LIN {X 0.236,Y -556.515,Z 1541.490,A 0.000,B 0.000,C 90.000,E1 124.199} C_DIS
LIN {X 0.231,Y -556.880,Z 1541.484,A 0.000,B 0.000,C 90.000,E1 123.086} C_DIS
LIN {X -0.003,Y -557.168,Z 1541.476,A 0.000,B 0.000,C 90.000,E1 121.720} C_DIS
LIN {X 0.132,Y -557.913,Z 1541.462,A 0.000,B 0.000,C 90.000,E1 119.205} C_DIS
LIN {X 0.047,Y -558.358,Z 1541.456,A 0.000,B 0.000,C 90.000,E1 118.103} C_DIS
LIN {X 0.056,Y -558.863,Z 1541.447,A 0.000,B 0.000,C 90.000,E1 116.437} C_DIS
LIN {X -0.021,Y -559.208,Z 1541.441,A 0.000,B 0.000,C 90.000,E1 115.335} C_DIS
LIN {X -0.037,Y -559.617,Z 1541.433,A 0.000,B 0.000,C 90.000,E1 113.951} C_DIS
LIN {X -0.269,Y -559.870,Z 1541.425,A 0.000,B 0.000,C 90.000,E1 112.589} C_DIS
LIN {X 0.126,Y -560.109,Z 1541.415,A 0.000,B 0.000,C 90.000,E1 110.610} C_DIS
LIN {X 0.134,Y -560.466,Z 1541.404,A 0.000,B 0.000,C 90.000,E1 108.671} C_DIS
LIN {X 0.145,Y -560.782,Z 1541.393,A 0.000,B 0.000,C 90.000,E1 106.732} C_DIS
LIN {X -0.026,Y -561.131,Z 1541.381,A 0.000,B 0.000,C 90.000,E1 104.537} C_DIS
LIN {X -0.171,Y -561.673,Z 1541.367,A 0.000,B 0.000,C 90.000,E1 102.063} C_DIS
LIN {X 0.022,Y -562.418,Z 1541.353,A 0.000,B 0.000,C 90.000,E1 99.557} C_DIS
LIN {X 0.312,Y -562.996,Z 1541.344,A 0.000,B 0.000,C 90.000,E1 97.871} C_DIS
LIN {X -0.187,Y -563.479,Z 1541.336,A 0.000,B 0.000,C 90.000,E1 96.543} C_DIS
LIN {X -0.081,Y -564.062,Z 1541.327,A 0.000,B 0.000,C 90.000,E1 94.878} C_DIS
LIN {X -0.053,Y -564.429,Z 1541.319,A 0.000,B 0.000,C 90.000,E1 93.498} C_DIS
LIN {X 0.057,Y -564.999,Z 1541.310,A 0.000,B 0.000,C 90.000,E1 91.835} C_DIS
LIN {X -0.161,Y -565.788,Z 1541.298,A 0.000,B 0.000,C 90.000,E1 89.656} C_DIS
LIN {X -0.247,Y -566.843,Z 1541.284,A 0.000,B 0.000,C 90.000,E1 87.192} C_DIS
LIN {X 0.050,Y -567.682,Z 1541.274,A 0.000,B 0.000,C 90.000,E1 85.241} C_DIS
LIN {X -0.107,Y -569.181,Z 1541.257,A 0.000,B 0.000,C 90.000,E1 82.243} C_DIS
LIN {X 0.052,Y -570.789,Z 1541.245,A 0.000,B 0.000,C 90.000,E1 80.038} C_DIS
LIN {X -0.035,Y -572.121,Z 1541.236,A 0.000,B 0.000,C 90.000,E1 78.409} C_DIS
LIN {X -0.018,Y -573.750,Z 1541.224,A 0.000,B 0.000,C 90.000,E1 76.228} C_DIS
LIN {X 0.006,Y -574.797,Z 1541.216,A 0.000,B 0.000,C 90.000,E1 74.866} C_DIS
LIN {X 0.042,Y -575.718,Z 1541.208,A 0.000,B 0.000,C 90.000,E1 73.504} C_DIS
LIN {X -0.285,Y -576.881,Z 1541.198,A 0.000,B 0.000,C 90.000,E1 71.638} C_DIS
LIN {X -0.015,Y -578.115,Z 1541.186,A 0.000,B 0.000,C 90.000,E1 69.444} C_DIS
LIN {X 0.256,Y -579.057,Z 1541.177,A 0.000,B 0.000,C 90.000,E1 67.794} C_DIS
LIN {X 0.079,Y -580.085,Z 1541.166,A 0.000,B 0.000,C 90.000,E1 65.921} C_DIS
LIN {X 0.030,Y -581.371,Z 1541.154,A 0.000,B 0.000,C 90.000,E1 63.768} C_DIS
LIN {X 0.017,Y -582.452,Z 1541.145,A 0.000,B 0.000,C 90.000,E1 62.153} C_DIS
LIN {X 0.153,Y -583.335,Z 1541.138,A 0.000,B 0.000,C 90.000,E1 60.795} C_DIS
LIN {X 0.080,Y -584.189,Z 1541.130,A 0.000,B 0.000,C 90.000,E1 59.459} C_DIS
LIN {X 0.028,Y -585.143,Z 1541.123,A 0.000,B 0.000,C 90.000,E1 58.122} C_DIS
LIN {X -0.019,Y -586.054,Z 1541.115,A 0.000,B 0.000,C 90.000,E1 56.786} C_DIS
LIN {X -0.084,Y -586.770,Z 1541.110,A 0.000,B 0.000,C 90.000,E1 55.722} C_DIS
LIN {X -0.271,Y -587.524,Z 1541.102,A 0.000,B 0.000,C 90.000,E1 54.402} C_DIS
LIN {X -0.107,Y -588.020,Z 1541.095,A 0.000,B 0.000,C 90.000,E1 53.050} C_DIS
LIN {X -0.203,Y -588.474,Z 1541.086,A 0.000,B 0.000,C 90.000,E1 51.457} C_DIS
LIN {X 0.134,Y -588.756,Z 1541.080,A 0.000,B 0.000,C 90.000,E1 50.356} C_DIS
LIN {X 0.273,Y -588.760,Z 1541.075,A 0.000,B 0.000,C 90.000,E1 49.542} C_DIS
LIN {X 0.215,Y -588.563,Z 1541.073,A 0.000,B 0.000,C 90.000,E1 49.013} C_DIS
LIN {X 0.155,Y -588.189,Z 1541.069,A 0.000,B 0.000,C 90.000,E1 48.485} C_DIS
LIN {X -0.095,Y -587.881,Z 1541.068,A 0.000,B 0.000,C 90.000,E1 48.243} C_DIS
LIN {X -0.160,Y -586.881,Z 1541.065,A 0.000,B 0.000,C 90.000,E1 47.715} C_DIS
LIN {X -0.014,Y -586.191,Z 1541.064,A 0.000,B 0.000,C 90.000,E1 47.433} C_DIS
LIN {X 0.165,Y -585.154,Z 1541.062,A 0.000,B 0.000,C 90.000,E1 47.148} C_DIS
LIN {X 0.054,Y -584.440,Z 1541.061,A 0.000,B 0.000,C 90.000,E1 47.025} C_DIS
LIN {X 0.031,Y -583.064,Z 1541.060,A 0.000,B 0.000,C 90.000,E1 46.863} C_DIS
LIN {X 0.138,Y -582.631,Z 1541.060,A 0.000,B 0.000,C 90.000,E1 46.824} C_DIS
LIN {X -0.118,Y -581.797,Z 1541.060,A 0.000,B 0.000,C 90.000,E1 46.824} C_DIS
LIN {X -0.127,Y -422.308,Z 1541.060,A 0.000,B 0.000,C 90.000,E1 46.824} C_DIS
LIN {X 0.122,Y -418.840,Z 1541.050,A 0.000,B 0.000,C 90.000,E1 44.919} C_DIS
LIN {X -0.221,Y -416.461,Z 1541.044,A 0.000,B 0.000,C 90.000,E1 43.947} C_DIS
LIN {X 0.118,Y -407.450,Z 1541.019,A 0.000,B 0.000,C 90.000,E1 39.439} C_DIS
LIN {X 0.243,Y -405.717,Z 1541.013,A 0.000,B 0.000,C 90.000,E1 38.382} C_DIS
LIN {X 0.206,Y -397.431,Z 1540.990,A 0.000,B 0.000,C 90.000,E1 34.199} C_DIS
LIN {X 0.070,Y -393.663,Z 1540.976,A 0.000,B 0.000,C 90.000,E1 31.750} C_DIS
LIN {X -0.160,Y -386.269,Z 1540.953,A 0.000,B 0.000,C 90.000,E1 27.513} C_DIS
LIN {X -0.001,Y -383.047,Z 1540.939,A 0.000,B 0.000,C 90.000,E1 24.975} C_DIS
LIN {X -0.032,Y -381.933,Z 1540.935,A 0.000,B 0.000,C 90.000,E1 24.259} C_DIS
LIN {X 0.090,Y -375.539,Z 1540.909,A 0.000,B 0.000,C 90.000,E1 19.523} C_DIS
LIN {X 0.085,Y -373.444,Z 1540.896,A 0.000,B 0.000,C 90.000,E1 17.330} C_DIS
LIN {X 0.018,Y -367.914,Z 1540.868,A 0.000,B 0.000,C 90.000,E1 12.187} C_DIS
LIN {X 0.037,Y -366.509,Z 1540.855,A 0.000,B 0.000,C 90.000,E1 9.962} C_DIS
LIN {X -0.027,Y -361.808,Z 1540.822,A 0.000,B 0.000,C 90.000,E1 4.012} C_DIS
LIN {X -0.142,Y -360.904,Z 1540.802,A 0.000,B 0.000,C 90.000,E1 0.286} C_DIS
LIN {X -0.053,Y -359.426,Z 1540.770,A 0.000,B 0.000,C 90.000,E1 354.546} C_DIS
LIN {X 0.070,Y -358.890,Z 1540.759,A 0.000,B 0.000,C 90.000,E1 352.648} C_DIS
LIN {X -0.020,Y -359.563,Z 1540.726,A 0.000,B 0.000,C 90.000,E1 346.645} C_DIS
LIN {X 0.001,Y -361.801,Z 1540.684,A 0.000,B 0.000,C 90.000,E1 339.135} C_DIS
LIN {X -0.154,Y -362.053,Z 1540.680,A 0.000,B 0.000,C 90.000,E1 338.411} C_DIS
LIN {X 0.189,Y -365.980,Z 1540.643,A 0.000,B 0.000,C 90.000,E1 331.641} C_DIS
LIN {X 0.029,Y -366.387,Z 1540.639,A 0.000,B 0.000,C 90.000,E1 330.923} C_DIS
LIN {X -0.031,Y -371.355,Z 1540.604,A 0.000,B 0.000,C 90.000,E1 324.642} C_DIS
LIN {X -0.043,Y -371.766,Z 1540.602,A 0.000,B 0.000,C 90.000,E1 324.276} C_DIS
LIN {X 0.013,Y -377.358,Z 1540.567,A 0.000,B 0.000,C 90.000,E1 318.038} C_DIS
LIN {X 0.012,Y -378.235,Z 1540.563,A 0.000,B 0.000,C 90.000,E1 317.310} C_DIS
LIN {X 0.002,Y -383.940,Z 1540.531,A 0.000,B 0.000,C 90.000,E1 311.515} C_DIS
LIN {X 0.088,Y -384.893,Z 1540.527,A 0.000,B 0.000,C 90.000,E1 310.782} C_DIS
LIN {X 0.262,Y -390.610,Z 1540.495,A 0.000,B 0.000,C 90.000,E1 305.025} C_DIS
LIN {X 0.106,Y -391.104,Z 1540.493,A 0.000,B 0.000,C 90.000,E1 304.692} C_DIS
LIN {X 0.022,Y -391.648,Z 1540.489,A 0.000,B 0.000,C 90.000,E1 303.992} C_DIS
LIN {X -0.080,Y -396.825,Z 1540.459,A 0.000,B 0.000,C 90.000,E1 298.693} C_DIS
LIN {X -0.210,Y -397.120,Z 1540.457,A 0.000,B 0.000,C 90.000,E1 298.359} C_DIS
LIN {X -0.055,Y -401.597,Z 1540.426,A 0.000,B 0.000,C 90.000,E1 292.717} C_DIS
LIN {X 0.222,Y -404.659,Z 1540.395,A 0.000,B 0.000,C 90.000,E1 287.094} C_DIS
LIN {X -0.079,Y -404.735,Z 1540.391,A 0.000,B 0.000,C 90.000,E1 286.441} C_DIS
LIN {X 0.214,Y -406.099,Z 1540.364,A 0.000,B 0.000,C 90.000,E1 281.535} C_DIS
LIN {X -0.176,Y -406.094,Z 1540.362,A 0.000,B 0.000,C 90.000,E1 281.243} C_DIS
LIN {X -0.097,Y -405.680,Z 1540.333,A 0.000,B 0.000,C 90.000,E1 276.024} C_DIS
LIN {X -0.165,Y -405.058,Z 1540.328,A 0.000,B 0.000,C 90.000,E1 274.992} C_DIS
LIN {X -0.060,Y -403.497,Z 1540.304,A 0.000,B 0.000,C 90.000,E1 270.802} C_DIS
LIN {X -0.092,Y -403.288,Z 1540.302,A 0.000,B 0.000,C 90.000,E1 270.458} C_DIS
LIN {X 0.091,Y -398.931,Z 1540.271,A 0.000,B 0.000,C 90.000,E1 264.837} C_DIS
LIN {X -0.040,Y -393.108,Z 1540.242,A 0.000,B 0.000,C 90.000,E1 259.567} C_DIS
LIN {X -0.079,Y -392.835,Z 1540.240,A 0.000,B 0.000,C 90.000,E1 259.218} C_DIS
LIN {X 0.034,Y -385.993,Z 1540.212,A 0.000,B 0.000,C 90.000,E1 254.212} C_DIS
LIN {X -0.026,Y -385.267,Z 1540.208,A 0.000,B 0.000,C 90.000,E1 253.504} C_DIS
LIN {X -0.004,Y -384.768,Z 1540.206,A 0.000,B 0.000,C 90.000,E1 253.142} C_DIS
LIN {X 0.221,Y -377.973,Z 1540.182,A 0.000,B 0.000,C 90.000,E1 248.773} C_DIS
LIN {X -0.044,Y -376.233,Z 1540.174,A 0.000,B 0.000,C 90.000,E1 247.358} C_DIS
LIN {X 0.057,Y -374.944,Z 1540.170,A 0.000,B 0.000,C 90.000,E1 246.613} C_DIS
LIN {X -0.208,Y -368.417,Z 1540.148,A 0.000,B 0.000,C 90.000,E1 242.615} C_DIS
LIN {X 0.097,Y -366.047,Z 1540.137,A 0.000,B 0.000,C 90.000,E1 240.717} C_DIS
LIN {X 0.004,Y -359.196,Z 1540.115,A 0.000,B 0.000,C 90.000,E1 236.628} C_DIS
LIN {X 0.021,Y -355.842,Z 1540.100,A 0.000,B 0.000,C 90.000,E1 233.989} C_DIS
LIN {X -0.173,Y -348.793,Z 1540.075,A 0.000,B 0.000,C 90.000,E1 229.461} C_DIS
LIN {X -0.097,Y -346.185,Z 1540.062,A 0.000,B 0.000,C 90.000,E1 227.148} C_DIS
LIN {X -0.088,Y -345.065,Z 1540.058,A 0.000,B 0.000,C 90.000,E1 226.377} C_DIS
LIN {X 0.094,Y -338.586,Z 1540.030,A 0.000,B 0.000,C 90.000,E1 221.310} C_DIS
LIN {X 0.094,Y -336.840,Z 1540.019,A 0.000,B 0.000,C 90.000,E1 219.358} C_DIS
LIN {X 0.014,Y -330.861,Z 1539.988,A 0.000,B 0.000,C 90.000,E1 213.865} C_DIS
LIN {X 0.149,Y -329.296,Z 1539.975,A 0.000,B 0.000,C 90.000,E1 211.465} C_DIS
LIN {X -0.154,Y -324.669,Z 1539.942,A 0.000,B 0.000,C 90.000,E1 205.540} C_DIS
LIN {X 0.174,Y -323.837,Z 1539.928,A 0.000,B 0.000,C 90.000,E1 203.078} C_DIS
LIN {X -0.017,Y -321.124,Z 1539.881,A 0.000,B 0.000,C 90.000,E1 194.662} C_DIS
LIN {X 0.138,Y -320.932,Z 1539.877,A 0.000,B 0.000,C 90.000,E1 193.828} C_DIS
LIN {X -0.076,Y -321.562,Z 1539.832,A 0.000,B 0.000,C 90.000,E1 185.796} C_DIS
LIN {X -0.143,Y -324.415,Z 1539.790,A 0.000,B 0.000,C 90.000,E1 178.165} C_DIS
LIN {X -0.141,Y -325.376,Z 1539.783,A 0.000,B 0.000,C 90.000,E1 176.963} C_DIS
LIN {X -0.100,Y -329.112,Z 1539.750,A 0.000,B 0.000,C 90.000,E1 170.971} C_DIS
LIN {X 0.061,Y -334.260,Z 1539.726,A 0.000,B 0.000,C 90.000,E1 166.589} C_DIS
LIN {X 0.067,Y -335.488,Z 1539.719,A 0.000,B 0.000,C 90.000,E1 165.408} C_DIS
LIN {X 0.143,Y -340.932,Z 1539.695,A 0.000,B 0.000,C 90.000,E1 161.094} C_DIS
LIN {X -0.172,Y -342.138,Z 1539.691,A 0.000,B 0.000,C 90.000,E1 160.369} C_DIS
LIN {X -0.058,Y -347.939,Z 1539.667,A 0.000,B 0.000,C 90.000,E1 156.102} C_DIS
LIN {X -0.081,Y -354.259,Z 1539.648,A 0.000,B 0.000,C 90.000,E1 152.666} C_DIS
LIN {X -0.222,Y -361.406,Z 1539.625,A 0.000,B 0.000,C 90.000,E1 148.535} C_DIS
LIN {X 0.065,Y -368.758,Z 1539.606,A 0.000,B 0.000,C 90.000,E1 145.135} C_DIS
LIN {X 0.065,Y -377.029,Z 1539.584,A 0.000,B 0.000,C 90.000,E1 141.090} C_DIS
LIN {X -0.061,Y -383.435,Z 1539.570,A 0.000,B 0.000,C 90.000,E1 138.566} C_DIS
LIN {X -0.015,Y -385.037,Z 1539.566,A 0.000,B 0.000,C 90.000,E1 137.838} C_DIS
LIN {X -0.004,Y -394.325,Z 1539.544,A 0.000,B 0.000,C 90.000,E1 133.905} C_DIS
LIN {X 0.107,Y -399.276,Z 1539.534,A 0.000,B 0.000,C 90.000,E1 132.123} C_DIS
LIN {X 0.210,Y -400.192,Z 1539.532,A 0.000,B 0.000,C 90.000,E1 131.757} C_DIS
LIN {X 0.078,Y -404.788,Z 1539.521,A 0.000,B 0.000,C 90.000,E1 129.806} C_DIS
LIN {X 0.058,Y -545.511,Z 1539.521,A 0.000,B 0.000,C 90.000,E1 129.806} C_DIS
LIN {X 0.013,Y -547.395,Z 1539.521,A 0.000,B 0.000,C 90.000,E1 129.688} C_DIS
LIN {X 0.033,Y -548.800,Z 1539.519,A 0.000,B 0.000,C 90.000,E1 129.483} C_DIS
LIN {X 0.077,Y -550.101,Z 1539.518,A 0.000,B 0.000,C 90.000,E1 129.197} C_DIS
LIN {X 0.131,Y -551.079,Z 1539.516,A 0.000,B 0.000,C 90.000,E1 128.910} C_DIS
LIN {X -0.186,Y -552.562,Z 1539.513,A 0.000,B 0.000,C 90.000,E1 128.382} C_DIS
LIN {X -0.060,Y -553.654,Z 1539.510,A 0.000,B 0.000,C 90.000,E1 127.810} C_DIS
LIN {X 0.151,Y -554.899,Z 1539.505,A 0.000,B 0.000,C 90.000,E1 126.950} C_DIS
LIN {X -0.074,Y -555.742,Z 1539.501,A 0.000,B 0.000,C 90.000,E1 126.137} C_DIS
LIN {X -0.093,Y -556.443,Z 1539.495,A 0.000,B 0.000,C 90.000,E1 125.025} C_DIS
LIN {X -0.100,Y -556.919,Z 1539.488,A 0.000,B 0.000,C 90.000,E1 123.913} C_DIS
LIN {X -0.177,Y -557.170,Z 1539.484,A 0.000,B 0.000,C 90.000,E1 123.086} C_DIS
LIN {X 0.067,Y -557.444,Z 1539.476,A 0.000,B 0.000,C 90.000,E1 121.671} C_DIS
LIN {X -0.049,Y -558.086,Z 1539.464,A 0.000,B 0.000,C 90.000,E1 119.461} C_DIS
LIN {X -0.344,Y -558.601,Z 1539.456,A 0.000,B 0.000,C 90.000,E1 118.103} C_DIS
LIN {X -0.081,Y -559.095,Z 1539.447,A 0.000,B 0.000,C 90.000,E1 116.411} C_DIS
LIN {X -0.103,Y -559.429,Z 1539.439,A 0.000,B 0.000,C 90.000,E1 115.027} C_DIS
LIN {X 0.094,Y -559.808,Z 1539.433,A 0.000,B 0.000,C 90.000,E1 113.898} C_DIS
LIN {X 0.086,Y -560.052,Z 1539.425,A 0.000,B 0.000,C 90.000,E1 112.514} C_DIS
LIN {X -0.246,Y -560.313,Z 1539.414,A 0.000,B 0.000,C 90.000,E1 110.610} C_DIS
LIN {X 0.170,Y -560.599,Z 1539.405,A 0.000,B 0.000,C 90.000,E1 108.906} C_DIS
LIN {X 0.018,Y -560.882,Z 1539.394,A 0.000,B 0.000,C 90.000,E1 106.985} C_DIS
LIN {X 0.111,Y -561.151,Z 1539.385,A 0.000,B 0.000,C 90.000,E1 105.315} C_DIS
LIN {X -0.235,Y -561.332,Z 1539.379,A 0.000,B 0.000,C 90.000,E1 104.245} C_DIS
LIN {X 0.026,Y -561.875,Z 1539.367,A 0.000,B 0.000,C 90.000,E1 102.007} C_DIS
LIN {X 0.073,Y -562.531,Z 1539.354,A 0.000,B 0.000,C 90.000,E1 99.792} C_DIS
LIN {X -0.185,Y -563.140,Z 1539.345,A 0.000,B 0.000,C 90.000,E1 98.163} C_DIS
LIN {X -0.118,Y -563.647,Z 1539.338,A 0.000,B 0.000,C 90.000,E1 96.777} C_DIS
LIN {X 0.148,Y -564.314,Z 1539.327,A 0.000,B 0.000,C 90.000,E1 94.821} C_DIS
LIN {X 0.182,Y -564.691,Z 1539.319,A 0.000,B 0.000,C 90.000,E1 93.440} C_DIS
LIN {X -0.249,Y -565.309,Z 1539.310,A 0.000,B 0.000,C 90.000,E1 91.833} C_DIS
LIN {X 0.089,Y -566.099,Z 1539.298,A 0.000,B 0.000,C 90.000,E1 89.599} C_DIS
LIN {X -0.102,Y -567.043,Z 1539.286,A 0.000,B 0.000,C 90.000,E1 87.421} C_DIS
LIN {X 0.093,Y -567.784,Z 1539.276,A 0.000,B 0.000,C 90.000,E1 85.755} C_DIS
LIN {X 0.188,Y -568.369,Z 1539.269,A 0.000,B 0.000,C 90.000,E1 84.375} C_DIS
LIN {X -0.212,Y -569.746,Z 1539.255,A 0.000,B 0.000,C 90.000,E1 81.951} C_DIS
LIN {X 0.060,Y -570.688,Z 1539.248,A 0.000,B 0.000,C 90.000,E1 80.557} C_DIS
LIN {X 0.160,Y -571.581,Z 1539.242,A 0.000,B 0.000,C 90.000,E1 79.454} C_DIS
LIN {X -0.107,Y -572.670,Z 1539.234,A 0.000,B 0.000,C 90.000,E1 78.117} C_DIS
LIN {X 0.283,Y -574.137,Z 1539.223,A 0.000,B 0.000,C 90.000,E1 76.172} C_DIS
LIN {X -0.244,Y -575.166,Z 1539.216,A 0.000,B 0.000,C 90.000,E1 74.866} C_DIS
LIN {X -0.201,Y -576.106,Z 1539.208,A 0.000,B 0.000,C 90.000,E1 73.504} C_DIS
LIN {X 0.028,Y -577.285,Z 1539.198,A 0.000,B 0.000,C 90.000,E1 71.583} C_DIS
LIN {X 0.303,Y -578.536,Z 1539.186,A 0.000,B 0.000,C 90.000,E1 69.390} C_DIS
LIN {X -0.107,Y -579.584,Z 1539.175,A 0.000,B 0.000,C 90.000,E1 67.539} C_DIS
LIN {X -0.267,Y -580.591,Z 1539.165,A 0.000,B 0.000,C 90.000,E1 65.665} C_DIS
LIN {X -0.166,Y -581.736,Z 1539.154,A 0.000,B 0.000,C 90.000,E1 63.768} C_DIS
LIN {X 0.213,Y -583.011,Z 1539.144,A 0.000,B 0.000,C 90.000,E1 61.847} C_DIS
LIN {X -0.002,Y -584.073,Z 1539.135,A 0.000,B 0.000,C 90.000,E1 60.255} C_DIS
LIN {X -0.318,Y -585.347,Z 1539.124,A 0.000,B 0.000,C 90.000,E1 58.408} C_DIS
LIN {X -0.046,Y -586.280,Z 1539.117,A 0.000,B 0.000,C 90.000,E1 57.041} C_DIS
LIN {X 0.243,Y -587.178,Z 1539.109,A 0.000,B 0.000,C 90.000,E1 55.674} C_DIS
LIN {X 0.055,Y -587.940,Z 1539.102,A 0.000,B 0.000,C 90.000,E1 54.356} C_DIS
LIN {X -0.251,Y -588.459,Z 1539.095,A 0.000,B 0.000,C 90.000,E1 53.050} C_DIS
LIN {X 0.122,Y -588.912,Z 1539.086,A 0.000,B 0.000,C 90.000,E1 51.412} C_DIS
LIN {X 0.149,Y -589.505,Z 1539.075,A 0.000,B 0.000,C 90.000,E1 49.542} C_DIS
LIN {X -0.153,Y -589.553,Z 1539.071,A 0.000,B 0.000,C 90.000,E1 48.771} C_DIS
LIN {X -0.205,Y -589.384,Z 1539.068,A 0.000,B 0.000,C 90.000,E1 48.243} C_DIS
LIN {X 0.327,Y -588.608,Z 1539.063,A 0.000,B 0.000,C 90.000,E1 47.391} C_DIS
LIN {X -0.165,Y -587.628,Z 1539.061,A 0.000,B 0.000,C 90.000,E1 46.905} C_DIS
LIN {X 0.016,Y -587.021,Z 1539.059,A 0.000,B 0.000,C 90.000,E1 46.620} C_DIS
LIN {X -0.233,Y -586.190,Z 1539.058,A 0.000,B 0.000,C 90.000,E1 46.377} C_DIS
LIN {X 0.344,Y -584.929,Z 1539.056,A 0.000,B 0.000,C 90.000,E1 46.053} C_DIS
LIN {X -0.274,Y -583.866,Z 1539.055,A 0.000,B 0.000,C 90.000,E1 45.972} C_DIS
LIN {X -0.132,Y -582.963,Z 1539.055,A 0.000,B 0.000,C 90.000,E1 45.891} C_DIS
LIN {X -0.362,Y -582.214,Z 1539.055,A 0.000,B 0.000,C 90.000,E1 45.891} C_DIS
LIN {X 0.017,Y -420.475,Z 1539.055,A 0.000,B 0.000,C 90.000,E1 45.850} C_DIS
LIN {X 0.032,Y -418.598,Z 1539.049,A 0.000,B 0.000,C 90.000,E1 44.798} C_DIS
LIN {X -0.163,Y -409.032,Z 1539.024,A 0.000,B 0.000,C 90.000,E1 40.378} C_DIS
LIN {X 0.020,Y -406.094,Z 1539.015,A 0.000,B 0.000,C 90.000,E1 38.624} C_DIS
LIN {X -0.124,Y -403.870,Z 1539.009,A 0.000,B 0.000,C 90.000,E1 37.604} C_DIS
LIN {X -0.031,Y -395.521,Z 1538.984,A 0.000,B 0.000,C 90.000,E1 33.038} C_DIS
LIN {X -0.211,Y -393.988,Z 1538.978,A 0.000,B 0.000,C 90.000,E1 32.005} C_DIS
LIN {X 0.059,Y -392.681,Z 1538.974,A 0.000,B 0.000,C 90.000,E1 31.258} C_DIS
LIN {X 0.100,Y -385.078,Z 1538.948,A 0.000,B 0.000,C 90.000,E1 26.616} C_DIS
LIN {X 0.068,Y -382.888,Z 1538.938,A 0.000,B 0.000,C 90.000,E1 24.823} C_DIS
LIN {X 0.014,Y -376.180,Z 1538.912,A 0.000,B 0.000,C 90.000,E1 20.120} C_DIS
LIN {X -0.117,Y -373.691,Z 1538.898,A 0.000,B 0.000,C 90.000,E1 17.583} C_DIS
LIN {X 0.018,Y -368.087,Z 1538.869,A 0.000,B 0.000,C 90.000,E1 12.411} C_DIS
LIN {X -0.174,Y -366.408,Z 1538.855,A 0.000,B 0.000,C 90.000,E1 9.849} C_DIS
LIN {X 0.125,Y -361.743,Z 1538.822,A 0.000,B 0.000,C 90.000,E1 3.841} C_DIS
LIN {X 0.011,Y -360.865,Z 1538.801,A 0.000,B 0.000,C 90.000,E1 0.115} C_DIS
LIN {X -0.053,Y -359.426,Z 1538.770,A 0.000,B 0.000,C 90.000,E1 354.546} C_DIS
LIN {X 0.070,Y -358.890,Z 1538.759,A 0.000,B 0.000,C 90.000,E1 352.648} C_DIS
LIN {X -0.020,Y -359.563,Z 1538.726,A 0.000,B 0.000,C 90.000,E1 346.645} C_DIS
LIN {X 0.001,Y -361.801,Z 1538.684,A 0.000,B 0.000,C 90.000,E1 339.135} C_DIS
LIN {X -0.154,Y -362.053,Z 1538.680,A 0.000,B 0.000,C 90.000,E1 338.411} C_DIS
LIN {X 0.189,Y -365.980,Z 1538.643,A 0.000,B 0.000,C 90.000,E1 331.641} C_DIS
LIN {X 0.029,Y -366.387,Z 1538.639,A 0.000,B 0.000,C 90.000,E1 330.923} C_DIS
LIN {X -0.031,Y -371.355,Z 1538.604,A 0.000,B 0.000,C 90.000,E1 324.642} C_DIS
LIN {X -0.043,Y -371.766,Z 1538.602,A 0.000,B 0.000,C 90.000,E1 324.276} C_DIS
LIN {X 0.013,Y -377.358,Z 1538.567,A 0.000,B 0.000,C 90.000,E1 318.038} C_DIS
LIN {X 0.012,Y -378.235,Z 1538.563,A 0.000,B 0.000,C 90.000,E1 317.310} C_DIS
LIN {X 0.002,Y -383.940,Z 1538.531,A 0.000,B 0.000,C 90.000,E1 311.515} C_DIS
LIN {X 0.088,Y -384.893,Z 1538.527,A 0.000,B 0.000,C 90.000,E1 310.782} C_DIS
LIN {X 0.262,Y -390.610,Z 1538.495,A 0.000,B 0.000,C 90.000,E1 305.025} C_DIS
LIN {X 0.106,Y -391.104,Z 1538.493,A 0.000,B 0.000,C 90.000,E1 304.692} C_DIS
LIN {X 0.022,Y -391.648,Z 1538.489,A 0.000,B 0.000,C 90.000,E1 303.992} C_DIS
LIN {X -0.080,Y -396.825,Z 1538.459,A 0.000,B 0.000,C 90.000,E1 298.693} C_DIS
LIN {X -0.210,Y -397.120,Z 1538.457,A 0.000,B 0.000,C 90.000,E1 298.359} C_DIS
LIN {X -0.055,Y -401.597,Z 1538.426,A 0.000,B 0.000,C 90.000,E1 292.717} C_DIS
LIN {X 0.222,Y -404.659,Z 1538.395,A 0.000,B 0.000,C 90.000,E1 287.094} C_DIS
LIN {X -0.079,Y -404.735,Z 1538.391,A 0.000,B 0.000,C 90.000,E1 286.441} C_DIS
LIN {X 0.214,Y -406.099,Z 1538.364,A 0.000,B 0.000,C 90.000,E1 281.535} C_DIS
LIN {X -0.176,Y -406.094,Z 1538.362,A 0.000,B 0.000,C 90.000,E1 281.243} C_DIS
LIN {X -0.097,Y -405.680,Z 1538.333,A 0.000,B 0.000,C 90.000,E1 276.024} C_DIS
LIN {X -0.165,Y -405.058,Z 1538.328,A 0.000,B 0.000,C 90.000,E1 274.992} C_DIS
LIN {X -0.060,Y -403.497,Z 1538.304,A 0.000,B 0.000,C 90.000,E1 270.802} C_DIS
LIN {X -0.092,Y -403.288,Z 1538.302,A 0.000,B 0.000,C 90.000,E1 270.458} C_DIS
LIN {X 0.091,Y -398.931,Z 1538.271,A 0.000,B 0.000,C 90.000,E1 264.837} C_DIS
LIN {X -0.040,Y -393.108,Z 1538.242,A 0.000,B 0.000,C 90.000,E1 259.567} C_DIS
LIN {X -0.079,Y -392.835,Z 1538.240,A 0.000,B 0.000,C 90.000,E1 259.218} C_DIS
LIN {X 0.034,Y -385.993,Z 1538.212,A 0.000,B 0.000,C 90.000,E1 254.212} C_DIS
LIN {X -0.026,Y -385.267,Z 1538.208,A 0.000,B 0.000,C 90.000,E1 253.504} C_DIS
LIN {X -0.004,Y -384.768,Z 1538.206,A 0.000,B 0.000,C 90.000,E1 253.142} C_DIS
LIN {X 0.221,Y -377.973,Z 1538.182,A 0.000,B 0.000,C 90.000,E1 248.773} C_DIS
LIN {X -0.044,Y -376.233,Z 1538.174,A 0.000,B 0.000,C 90.000,E1 247.358} C_DIS
LIN {X 0.057,Y -374.944,Z 1538.170,A 0.000,B 0.000,C 90.000,E1 246.613} C_DIS
LIN {X -0.208,Y -368.417,Z 1538.148,A 0.000,B 0.000,C 90.000,E1 242.615} C_DIS
LIN {X 0.097,Y -366.047,Z 1538.137,A 0.000,B 0.000,C 90.000,E1 240.717} C_DIS
LIN {X 0.004,Y -359.196,Z 1538.115,A 0.000,B 0.000,C 90.000,E1 236.628} C_DIS
LIN {X 0.021,Y -355.842,Z 1538.100,A 0.000,B 0.000,C 90.000,E1 233.989} C_DIS
LIN {X -0.173,Y -348.793,Z 1538.075,A 0.000,B 0.000,C 90.000,E1 229.461} C_DIS
LIN {X -0.097,Y -346.185,Z 1538.062,A 0.000,B 0.000,C 90.000,E1 227.148} C_DIS
LIN {X -0.088,Y -345.065,Z 1538.058,A 0.000,B 0.000,C 90.000,E1 226.377} C_DIS
LIN {X 0.094,Y -338.586,Z 1538.030,A 0.000,B 0.000,C 90.000,E1 221.310} C_DIS
LIN {X 0.094,Y -336.840,Z 1538.019,A 0.000,B 0.000,C 90.000,E1 219.358} C_DIS
LIN {X 0.014,Y -330.861,Z 1537.988,A 0.000,B 0.000,C 90.000,E1 213.865} C_DIS
LIN {X 0.149,Y -329.296,Z 1537.975,A 0.000,B 0.000,C 90.000,E1 211.465} C_DIS
LIN {X -0.154,Y -324.669,Z 1537.942,A 0.000,B 0.000,C 90.000,E1 205.540} C_DIS
LIN {X 0.174,Y -323.837,Z 1537.928,A 0.000,B 0.000,C 90.000,E1 203.078} C_DIS
LIN {X -0.017,Y -321.124,Z 1537.881,A 0.000,B 0.000,C 90.000,E1 194.662} C_DIS
LIN {X 0.138,Y -320.932,Z 1537.877,A 0.000,B 0.000,C 90.000,E1 193.828} C_DIS
LIN {X -0.076,Y -321.562,Z 1537.832,A 0.000,B 0.000,C 90.000,E1 185.796} C_DIS
LIN {X -0.143,Y -324.415,Z 1537.790,A 0.000,B 0.000,C 90.000,E1 178.165} C_DIS
LIN {X -0.141,Y -325.376,Z 1537.783,A 0.000,B 0.000,C 90.000,E1 176.963} C_DIS
LIN {X -0.100,Y -329.112,Z 1537.750,A 0.000,B 0.000,C 90.000,E1 170.971} C_DIS
LIN {X 0.061,Y -334.260,Z 1537.726,A 0.000,B 0.000,C 90.000,E1 166.589} C_DIS
LIN {X 0.067,Y -335.488,Z 1537.719,A 0.000,B 0.000,C 90.000,E1 165.408} C_DIS
LIN {X 0.143,Y -340.932,Z 1537.695,A 0.000,B 0.000,C 90.000,E1 161.094} C_DIS
LIN {X -0.172,Y -342.138,Z 1537.691,A 0.000,B 0.000,C 90.000,E1 160.369} C_DIS
LIN {X -0.058,Y -347.939,Z 1537.667,A 0.000,B 0.000,C 90.000,E1 156.102} C_DIS
LIN {X -0.081,Y -354.259,Z 1537.648,A 0.000,B 0.000,C 90.000,E1 152.666} C_DIS
LIN {X -0.222,Y -361.406,Z 1537.625,A 0.000,B 0.000,C 90.000,E1 148.535} C_DIS
LIN {X 0.065,Y -368.758,Z 1537.606,A 0.000,B 0.000,C 90.000,E1 145.135} C_DIS
LIN {X 0.065,Y -377.029,Z 1537.584,A 0.000,B 0.000,C 90.000,E1 141.090} C_DIS
LIN {X -0.061,Y -383.435,Z 1537.570,A 0.000,B 0.000,C 90.000,E1 138.566} C_DIS
LIN {X -0.015,Y -385.037,Z 1537.566,A 0.000,B 0.000,C 90.000,E1 137.838} C_DIS
LIN {X -0.004,Y -394.325,Z 1537.544,A 0.000,B 0.000,C 90.000,E1 133.905} C_DIS
LIN {X 0.107,Y -399.276,Z 1537.534,A 0.000,B 0.000,C 90.000,E1 132.123} C_DIS
LIN {X 0.210,Y -400.192,Z 1537.532,A 0.000,B 0.000,C 90.000,E1 131.757} C_DIS
LIN {X 0.170,Y -402.407,Z 1537.527,A 0.000,B 0.000,C 90.000,E1 130.782} C_DIS
LIN {X 0.184,Y -545.069,Z 1537.527,A 0.000,B 0.000,C 90.000,E1 130.782} C_DIS
LIN {X -0.074,Y -546.344,Z 1537.526,A 0.000,B 0.000,C 90.000,E1 130.744} C_DIS
LIN {X 0.279,Y -547.774,Z 1537.525,A 0.000,B 0.000,C 90.000,E1 130.539} C_DIS
LIN {X -0.102,Y -549.264,Z 1537.524,A 0.000,B 0.000,C 90.000,E1 130.297} C_DIS
LIN {X -0.056,Y -550.353,Z 1537.522,A 0.000,B 0.000,C 90.000,E1 130.011} C_DIS
LIN {X 0.049,Y -551.991,Z 1537.519,A 0.000,B 0.000,C 90.000,E1 129.439} C_DIS
LIN {X -0.258,Y -553.192,Z 1537.516,A 0.000,B 0.000,C 90.000,E1 128.910} C_DIS
LIN {X 0.218,Y -554.105,Z 1537.513,A 0.000,B 0.000,C 90.000,E1 128.302} C_DIS
LIN {X -0.348,Y -555.111,Z 1537.508,A 0.000,B 0.000,C 90.000,E1 127.523} C_DIS
LIN {X -0.122,Y -555.810,Z 1537.504,A 0.000,B 0.000,C 90.000,E1 126.664} C_DIS
LIN {X 0.267,Y -556.618,Z 1537.496,A 0.000,B 0.000,C 90.000,E1 125.231} C_DIS
LIN {X 0.264,Y -557.134,Z 1537.490,A 0.000,B 0.000,C 90.000,E1 124.119} C_DIS
LIN {X -0.039,Y -557.444,Z 1537.484,A 0.000,B 0.000,C 90.000,E1 123.038} C_DIS
LIN {X -0.258,Y -557.714,Z 1537.476,A 0.000,B 0.000,C 90.000,E1 121.671} C_DIS
LIN {X 0.119,Y -558.326,Z 1537.464,A 0.000,B 0.000,C 90.000,E1 119.411} C_DIS
LIN {X 0.098,Y -558.808,Z 1537.456,A 0.000,B 0.000,C 90.000,E1 118.025} C_DIS
LIN {X -0.185,Y -559.217,Z 1537.448,A 0.000,B 0.000,C 90.000,E1 116.668} C_DIS
LIN {X -0.205,Y -559.557,Z 1537.440,A 0.000,B 0.000,C 90.000,E1 115.283} C_DIS
LIN {X -0.210,Y -559.953,Z 1537.433,A 0.000,B 0.000,C 90.000,E1 113.898} C_DIS
LIN {X 0.094,Y -560.194,Z 1537.423,A 0.000,B 0.000,C 90.000,E1 112.206} C_DIS
LIN {X -0.020,Y -560.460,Z 1537.414,A 0.000,B 0.000,C 90.000,E1 110.556} C_DIS
LIN {X -0.124,Y -560.744,Z 1537.405,A 0.000,B 0.000,C 90.000,E1 108.906} C_DIS
LIN {X -0.110,Y -561.024,Z 1537.394,A 0.000,B 0.000,C 90.000,E1 106.968} C_DIS
LIN {X -0.028,Y -561.307,Z 1537.385,A 0.000,B 0.000,C 90.000,E1 105.300} C_DIS
LIN {X 0.311,Y -561.530,Z 1537.377,A 0.000,B 0.000,C 90.000,E1 103.883} C_DIS
LIN {X -0.255,Y -562.049,Z 1537.367,A 0.000,B 0.000,C 90.000,E1 102.007} C_DIS
LIN {X 0.291,Y -562.650,Z 1537.356,A 0.000,B 0.000,C 90.000,E1 100.018} C_DIS
LIN {X 0.100,Y -563.339,Z 1537.345,A 0.000,B 0.000,C 90.000,E1 98.106} C_DIS
LIN {X 0.087,Y -563.800,Z 1537.339,A 0.000,B 0.000,C 90.000,E1 97.004} C_DIS
LIN {X -0.214,Y -564.471,Z 1537.328,A 0.000,B 0.000,C 90.000,E1 95.106} C_DIS
LIN {X -0.183,Y -564.873,Z 1537.321,A 0.000,B 0.000,C 90.000,E1 93.726} C_DIS
LIN {X 0.063,Y -565.591,Z 1537.310,A 0.000,B 0.000,C 90.000,E1 91.776} C_DIS
LIN {X -0.272,Y -566.295,Z 1537.299,A 0.000,B 0.000,C 90.000,E1 89.885} C_DIS
LIN {X -0.141,Y -566.973,Z 1537.290,A 0.000,B 0.000,C 90.000,E1 88.224} C_DIS
LIN {X 0.043,Y -567.751,Z 1537.281,A 0.000,B 0.000,C 90.000,E1 86.560} C_DIS
LIN {X 0.252,Y -568.524,Z 1537.272,A 0.000,B 0.000,C 90.000,E1 84.894} C_DIS
LIN {X -0.039,Y -569.304,Z 1537.263,A 0.000,B 0.000,C 90.000,E1 83.280} C_DIS
LIN {X -0.240,Y -570.302,Z 1537.254,A 0.000,B 0.000,C 90.000,E1 81.659} C_DIS
LIN {X -0.145,Y -571.037,Z 1537.248,A 0.000,B 0.000,C 90.000,E1 80.557} C_DIS
LIN {X 0.152,Y -572.166,Z 1537.240,A 0.000,B 0.000,C 90.000,E1 79.162} C_DIS
LIN {X 0.015,Y -573.223,Z 1537.232,A 0.000,B 0.000,C 90.000,E1 77.813} C_DIS
LIN {X -0.260,Y -574.728,Z 1537.222,A 0.000,B 0.000,C 90.000,E1 75.936} C_DIS
LIN {X -0.223,Y -575.725,Z 1537.214,A 0.000,B 0.000,C 90.000,E1 74.574} C_DIS
LIN {X -0.011,Y -576.615,Z 1537.207,A 0.000,B 0.000,C 90.000,E1 73.196} C_DIS
LIN {X -0.138,Y -577.679,Z 1537.198,A 0.000,B 0.000,C 90.000,E1 71.583} C_DIS
LIN {X 0.149,Y -578.945,Z 1537.186,A 0.000,B 0.000,C 90.000,E1 69.390} C_DIS
LIN {X -0.252,Y -579.969,Z 1537.175,A 0.000,B 0.000,C 90.000,E1 67.539} C_DIS
LIN {X 0.126,Y -580.961,Z 1537.165,A 0.000,B 0.000,C 90.000,E1 65.613} C_DIS
LIN {X -0.294,Y -582.091,Z 1537.154,A 0.000,B 0.000,C 90.000,E1 63.768} C_DIS
LIN {X 0.094,Y -583.361,Z 1537.144,A 0.000,B 0.000,C 90.000,E1 61.847} C_DIS
LIN {X -0.241,Y -584.632,Z 1537.133,A 0.000,B 0.000,C 90.000,E1 59.999} C_DIS
LIN {X -0.113,Y -585.736,Z 1537.124,A 0.000,B 0.000,C 90.000,E1 58.377} C_DIS
LIN {X -0.142,Y -586.647,Z 1537.117,A 0.000,B 0.000,C 90.000,E1 57.041} C_DIS
LIN {X 0.347,Y -587.744,Z 1537.108,A 0.000,B 0.000,C 90.000,E1 55.388} C_DIS
LIN {X -0.028,Y -588.329,Z 1537.102,A 0.000,B 0.000,C 90.000,E1 54.356} C_DIS
LIN {X 0.144,Y -588.896,Z 1537.095,A 0.000,B 0.000,C 90.000,E1 53.004} C_DIS
LIN {X -0.145,Y -589.270,Z 1537.087,A 0.000,B 0.000,C 90.000,E1 51.698} C_DIS
LIN {X 0.093,Y -589.951,Z 1537.075,A 0.000,B 0.000,C 90.000,E1 49.542} C_DIS
LIN {X -0.007,Y -590.263,Z 1537.069,A 0.000,B 0.000,C 90.000,E1 48.485} C_DIS
LIN {X 0.096,Y -590.100,Z 1537.065,A 0.000,B 0.000,C 90.000,E1 47.676} C_DIS
LIN {X 0.047,Y -589.725,Z 1537.062,A 0.000,B 0.000,C 90.000,E1 47.148} C_DIS
LIN {X -0.008,Y -589.195,Z 1537.059,A 0.000,B 0.000,C 90.000,E1 46.620} C_DIS
LIN {X 0.337,Y -588.311,Z 1537.056,A 0.000,B 0.000,C 90.000,E1 46.053} C_DIS
LIN {X 0.092,Y -587.677,Z 1537.055,A 0.000,B 0.000,C 90.000,E1 45.810} C_DIS
LIN {X -0.154,Y -586.839,Z 1537.053,A 0.000,B 0.000,C 90.000,E1 45.567} C_DIS
LIN {X 0.016,Y -585.707,Z 1537.052,A 0.000,B 0.000,C 90.000,E1 45.283} C_DIS
LIN {X -0.111,Y -584.929,Z 1537.051,A 0.000,B 0.000,C 90.000,E1 45.162} C_DIS
LIN {X 0.178,Y -583.799,Z 1537.050,A 0.000,B 0.000,C 90.000,E1 45.000} C_DIS
LIN {X -0.006,Y -582.897,Z 1537.050,A 0.000,B 0.000,C 90.000,E1 44.960} C_DIS
LIN {X 0.248,Y -582.358,Z 1537.050,A 0.000,B 0.000,C 90.000,E1 44.919} C_DIS
LIN {X 0.156,Y -418.849,Z 1537.050,A 0.000,B 0.000,C 90.000,E1 44.919} C_DIS
LIN {X -0.170,Y -417.642,Z 1537.047,A 0.000,B 0.000,C 90.000,E1 44.433} C_DIS
LIN {X 0.184,Y -408.317,Z 1537.022,A 0.000,B 0.000,C 90.000,E1 39.930} C_DIS
LIN {X -0.109,Y -406.009,Z 1537.014,A 0.000,B 0.000,C 90.000,E1 38.588} C_DIS
LIN {X -0.129,Y -397.699,Z 1536.991,A 0.000,B 0.000,C 90.000,E1 34.405} C_DIS
LIN {X -0.047,Y -393.913,Z 1536.977,A 0.000,B 0.000,C 90.000,E1 31.926} C_DIS
LIN {X 0.063,Y -386.503,Z 1536.954,A 0.000,B 0.000,C 90.000,E1 27.641} C_DIS
LIN {X 0.040,Y -382.814,Z 1536.938,A 0.000,B 0.000,C 90.000,E1 24.771} C_DIS
LIN {X -0.006,Y -376.116,Z 1536.911,A 0.000,B 0.000,C 90.000,E1 20.066} C_DIS
LIN {X -0.021,Y -373.644,Z 1536.897,A 0.000,B 0.000,C 90.000,E1 17.511} C_DIS
LIN {X 0.008,Y -368.042,Z 1536.869,A 0.000,B 0.000,C 90.000,E1 12.355} C_DIS
LIN {X -0.120,Y -366.344,Z 1536.854,A 0.000,B 0.000,C 90.000,E1 9.782} C_DIS
LIN {X 0.118,Y -361.717,Z 1536.821,A 0.000,B 0.000,C 90.000,E1 3.784} C_DIS
LIN {X 0.004,Y -360.831,Z 1536.800,A 0.000,B 0.000,C 90.000,E1 0.057} C_DIS
LIN {X -0.053,Y -359.426,Z 1536.770,A 0.000,B 0.000,C 90.000,E1 354.546} C_DIS
LIN {X 0.070,Y -358.890,Z 1536.759,A 0.000,B 0.000,C 90.000,E1 352.648} C_DIS
LIN {X -0.020,Y -359.563,Z 1536.726,A 0.000,B 0.000,C 90.000,E1 346.645} C_DIS
LIN {X 0.001,Y -361.801,Z 1536.684,A 0.000,B 0.000,C 90.000,E1 339.135} C_DIS
LIN {X -0.154,Y -362.053,Z 1536.680,A 0.000,B 0.000,C 90.000,E1 338.411} C_DIS
LIN {X 0.189,Y -365.980,Z 1536.643,A 0.000,B 0.000,C 90.000,E1 331.641} C_DIS
LIN {X 0.029,Y -366.387,Z 1536.639,A 0.000,B 0.000,C 90.000,E1 330.923} C_DIS
LIN {X -0.031,Y -371.355,Z 1536.604,A 0.000,B 0.000,C 90.000,E1 324.642} C_DIS
LIN {X -0.043,Y -371.766,Z 1536.602,A 0.000,B 0.000,C 90.000,E1 324.276} C_DIS
LIN {X 0.013,Y -377.358,Z 1536.567,A 0.000,B 0.000,C 90.000,E1 318.038} C_DIS
LIN {X 0.012,Y -378.235,Z 1536.563,A 0.000,B 0.000,C 90.000,E1 317.310} C_DIS
LIN {X 0.002,Y -383.940,Z 1536.531,A 0.000,B 0.000,C 90.000,E1 311.515} C_DIS
LIN {X 0.088,Y -384.893,Z 1536.527,A 0.000,B 0.000,C 90.000,E1 310.782} C_DIS
LIN {X 0.262,Y -390.610,Z 1536.495,A 0.000,B 0.000,C 90.000,E1 305.025} C_DIS
LIN {X 0.106,Y -391.104,Z 1536.493,A 0.000,B 0.000,C 90.000,E1 304.692} C_DIS
LIN {X 0.022,Y -391.648,Z 1536.489,A 0.000,B 0.000,C 90.000,E1 303.992} C_DIS
LIN {X -0.080,Y -396.825,Z 1536.459,A 0.000,B 0.000,C 90.000,E1 298.693} C_DIS
LIN {X -0.210,Y -397.120,Z 1536.457,A 0.000,B 0.000,C 90.000,E1 298.359} C_DIS
LIN {X -0.055,Y -401.597,Z 1536.426,A 0.000,B 0.000,C 90.000,E1 292.717} C_DIS
LIN {X 0.222,Y -404.659,Z 1536.395,A 0.000,B 0.000,C 90.000,E1 287.094} C_DIS
LIN {X -0.079,Y -404.735,Z 1536.391,A 0.000,B 0.000,C 90.000,E1 286.441} C_DIS
LIN {X 0.214,Y -406.099,Z 1536.364,A 0.000,B 0.000,C 90.000,E1 281.535} C_DIS
LIN {X -0.176,Y -406.094,Z 1536.362,A 0.000,B 0.000,C 90.000,E1 281.243} C_DIS
LIN {X -0.097,Y -405.680,Z 1536.333,A 0.000,B 0.000,C 90.000,E1 276.024} C_DIS
LIN {X -0.165,Y -405.058,Z 1536.328,A 0.000,B 0.000,C 90.000,E1 274.992} C_DIS
LIN {X -0.060,Y -403.497,Z 1536.304,A 0.000,B 0.000,C 90.000,E1 270.802} C_DIS
LIN {X -0.092,Y -403.288,Z 1536.302,A 0.000,B 0.000,C 90.000,E1 270.458} C_DIS
LIN {X 0.091,Y -398.931,Z 1536.271,A 0.000,B 0.000,C 90.000,E1 264.837} C_DIS
LIN {X -0.040,Y -393.108,Z 1536.242,A 0.000,B 0.000,C 90.000,E1 259.567} C_DIS
LIN {X -0.079,Y -392.835,Z 1536.240,A 0.000,B 0.000,C 90.000,E1 259.218} C_DIS
LIN {X 0.034,Y -385.993,Z 1536.212,A 0.000,B 0.000,C 90.000,E1 254.212} C_DIS
LIN {X -0.026,Y -385.267,Z 1536.208,A 0.000,B 0.000,C 90.000,E1 253.504} C_DIS
LIN {X -0.004,Y -384.768,Z 1536.206,A 0.000,B 0.000,C 90.000,E1 253.142} C_DIS
LIN {X 0.221,Y -377.973,Z 1536.182,A 0.000,B 0.000,C 90.000,E1 248.773} C_DIS
LIN {X -0.044,Y -376.233,Z 1536.174,A 0.000,B 0.000,C 90.000,E1 247.358} C_DIS
LIN {X 0.057,Y -374.944,Z 1536.170,A 0.000,B 0.000,C 90.000,E1 246.613} C_DIS
LIN {X -0.208,Y -368.417,Z 1536.148,A 0.000,B 0.000,C 90.000,E1 242.615} C_DIS
LIN {X 0.097,Y -366.047,Z 1536.137,A 0.000,B 0.000,C 90.000,E1 240.717} C_DIS
LIN {X 0.004,Y -359.196,Z 1536.115,A 0.000,B 0.000,C 90.000,E1 236.628} C_DIS
LIN {X 0.021,Y -355.842,Z 1536.100,A 0.000,B 0.000,C 90.000,E1 233.989} C_DIS
LIN {X -0.173,Y -348.793,Z 1536.075,A 0.000,B 0.000,C 90.000,E1 229.461} C_DIS
LIN {X -0.097,Y -346.185,Z 1536.062,A 0.000,B 0.000,C 90.000,E1 227.148} C_DIS
LIN {X -0.088,Y -345.065,Z 1536.058,A 0.000,B 0.000,C 90.000,E1 226.377} C_DIS
LIN {X 0.094,Y -338.586,Z 1536.030,A 0.000,B 0.000,C 90.000,E1 221.310} C_DIS
LIN {X 0.094,Y -336.840,Z 1536.019,A 0.000,B 0.000,C 90.000,E1 219.358} C_DIS
LIN {X 0.014,Y -330.861,Z 1535.988,A 0.000,B 0.000,C 90.000,E1 213.865} C_DIS
LIN {X 0.149,Y -329.296,Z 1535.975,A 0.000,B 0.000,C 90.000,E1 211.465} C_DIS
LIN {X -0.154,Y -324.669,Z 1535.942,A 0.000,B 0.000,C 90.000,E1 205.540} C_DIS
LIN {X 0.174,Y -323.837,Z 1535.928,A 0.000,B 0.000,C 90.000,E1 203.078} C_DIS
LIN {X -0.017,Y -321.124,Z 1535.881,A 0.000,B 0.000,C 90.000,E1 194.662} C_DIS
LIN {X 0.138,Y -320.932,Z 1535.877,A 0.000,B 0.000,C 90.000,E1 193.828} C_DIS
LIN {X -0.076,Y -321.562,Z 1535.832,A 0.000,B 0.000,C 90.000,E1 185.796} C_DIS
LIN {X -0.143,Y -324.415,Z 1535.790,A 0.000,B 0.000,C 90.000,E1 178.165} C_DIS
LIN {X -0.141,Y -325.376,Z 1535.783,A 0.000,B 0.000,C 90.000,E1 176.963} C_DIS
LIN {X -0.100,Y -329.112,Z 1535.750,A 0.000,B 0.000,C 90.000,E1 170.971} C_DIS
LIN {X 0.061,Y -334.260,Z 1535.726,A 0.000,B 0.000,C 90.000,E1 166.589} C_DIS
LIN {X 0.067,Y -335.488,Z 1535.719,A 0.000,B 0.000,C 90.000,E1 165.408} C_DIS
LIN {X 0.143,Y -340.932,Z 1535.695,A 0.000,B 0.000,C 90.000,E1 161.094} C_DIS
LIN {X -0.172,Y -342.138,Z 1535.691,A 0.000,B 0.000,C 90.000,E1 160.369} C_DIS
LIN {X -0.058,Y -347.939,Z 1535.667,A 0.000,B 0.000,C 90.000,E1 156.102} C_DIS
LIN {X -0.081,Y -354.259,Z 1535.648,A 0.000,B 0.000,C 90.000,E1 152.666} C_DIS
LIN {X -0.222,Y -361.406,Z 1535.625,A 0.000,B 0.000,C 90.000,E1 148.535} C_DIS
LIN {X 0.065,Y -368.758,Z 1535.606,A 0.000,B 0.000,C 90.000,E1 145.135} C_DIS
LIN {X 0.065,Y -377.029,Z 1535.584,A 0.000,B 0.000,C 90.000,E1 141.090} C_DIS
LIN {X -0.061,Y -383.435,Z 1535.570,A 0.000,B 0.000,C 90.000,E1 138.566} C_DIS
LIN {X -0.015,Y -385.037,Z 1535.566,A 0.000,B 0.000,C 90.000,E1 137.838} C_DIS
LIN {X -0.004,Y -394.325,Z 1535.544,A 0.000,B 0.000,C 90.000,E1 133.905} C_DIS
LIN {X 0.107,Y -399.276,Z 1535.534,A 0.000,B 0.000,C 90.000,E1 132.123} C_DIS
LIN {X 0.141,Y -400.214,Z 1535.532,A 0.000,B 0.000,C 90.000,E1 131.757} C_DIS
LIN {X 0.160,Y -544.511,Z 1535.532,A 0.000,B 0.000,C 90.000,E1 131.757} C_DIS
LIN {X 0.066,Y -544.934,Z 1535.532,A 0.000,B 0.000,C 90.000,E1 131.757} C_DIS
LIN {X 0.047,Y -546.939,Z 1535.531,A 0.000,B 0.000,C 90.000,E1 131.595} C_DIS
LIN {X 0.026,Y -548.009,Z 1535.530,A 0.000,B 0.000,C 90.000,E1 131.434} C_DIS
LIN {X 0.063,Y -549.303,Z 1535.529,A 0.000,B 0.000,C 90.000,E1 131.148} C_DIS
LIN {X 0.108,Y -550.278,Z 1535.527,A 0.000,B 0.000,C 90.000,E1 130.862} C_DIS
LIN {X 0.148,Y -551.807,Z 1535.524,A 0.000,B 0.000,C 90.000,E1 130.297} C_DIS
LIN {X 0.262,Y -552.970,Z 1535.521,A 0.000,B 0.000,C 90.000,E1 129.725} C_DIS
LIN {X -0.038,Y -553.913,Z 1535.518,A 0.000,B 0.000,C 90.000,E1 129.197} C_DIS
LIN {X -0.264,Y -554.894,Z 1535.513,A 0.000,B 0.000,C 90.000,E1 128.382} C_DIS
LIN {X 0.034,Y -555.727,Z 1535.507,A 0.000,B 0.000,C 90.000,E1 127.237} C_DIS
LIN {X -0.104,Y -556.451,Z 1535.501,A 0.000,B 0.000,C 90.000,E1 126.137} C_DIS
LIN {X -0.112,Y -557.041,Z 1535.495,A 0.000,B 0.000,C 90.000,E1 125.025} C_DIS
LIN {X -0.109,Y -557.478,Z 1535.488,A 0.000,B 0.000,C 90.000,E1 123.913} C_DIS
LIN {X -0.105,Y -557.762,Z 1535.482,A 0.000,B 0.000,C 90.000,E1 122.801} C_DIS
LIN {X 0.146,Y -558.013,Z 1535.474,A 0.000,B 0.000,C 90.000,E1 121.386} C_DIS
LIN {X -0.030,Y -558.565,Z 1535.464,A 0.000,B 0.000,C 90.000,E1 119.461} C_DIS
LIN {X 0.026,Y -559.164,Z 1535.453,A 0.000,B 0.000,C 90.000,E1 117.513} C_DIS
LIN {X 0.251,Y -559.515,Z 1535.445,A 0.000,B 0.000,C 90.000,E1 116.104} C_DIS
LIN {X -0.165,Y -560.009,Z 1535.434,A 0.000,B 0.000,C 90.000,E1 114.207} C_DIS
LIN {X 0.139,Y -560.304,Z 1535.425,A 0.000,B 0.000,C 90.000,E1 112.514} C_DIS
LIN {X 0.027,Y -560.554,Z 1535.416,A 0.000,B 0.000,C 90.000,E1 110.865} C_DIS
LIN {X 0.238,Y -560.890,Z 1535.405,A 0.000,B 0.000,C 90.000,E1 108.906} C_DIS
LIN {X 0.091,Y -561.186,Z 1535.394,A 0.000,B 0.000,C 90.000,E1 106.985} C_DIS
LIN {X 0.192,Y -561.448,Z 1535.385,A 0.000,B 0.000,C 90.000,E1 105.315} C_DIS
LIN {X -0.106,Y -561.826,Z 1535.375,A 0.000,B 0.000,C 90.000,E1 103.411} C_DIS
LIN {X -0.274,Y -562.276,Z 1535.365,A 0.000,B 0.000,C 90.000,E1 101.771} C_DIS
LIN {X 0.117,Y -562.843,Z 1535.356,A 0.000,B 0.000,C 90.000,E1 100.074} C_DIS
LIN {X -0.073,Y -563.516,Z 1535.345,A 0.000,B 0.000,C 90.000,E1 98.163} C_DIS
LIN {X 0.002,Y -564.098,Z 1535.338,A 0.000,B 0.000,C 90.000,E1 96.777} C_DIS
LIN {X -0.284,Y -564.773,Z 1535.327,A 0.000,B 0.000,C 90.000,E1 94.878} C_DIS
LIN {X 0.004,Y -565.401,Z 1535.316,A 0.000,B 0.000,C 90.000,E1 92.922} C_DIS
LIN {X 0.127,Y -566.049,Z 1535.307,A 0.000,B 0.000,C 90.000,E1 91.260} C_DIS
LIN {X 0.256,Y -566.681,Z 1535.298,A 0.000,B 0.000,C 90.000,E1 89.599} C_DIS
LIN {X -0.155,Y -567.396,Z 1535.289,A 0.000,B 0.000,C 90.000,E1 87.993} C_DIS
LIN {X 0.017,Y -568.176,Z 1535.280,A 0.000,B 0.000,C 90.000,E1 86.331} C_DIS
LIN {X 0.231,Y -568.984,Z 1535.271,A 0.000,B 0.000,C 90.000,E1 84.666} C_DIS
LIN {X -0.058,Y -569.798,Z 1535.261,A 0.000,B 0.000,C 90.000,E1 83.053} C_DIS
LIN {X -0.257,Y -570.819,Z 1535.252,A 0.000,B 0.000,C 90.000,E1 81.432} C_DIS
LIN {X 0.215,Y -571.338,Z 1535.248,A 0.000,B 0.000,C 90.000,E1 80.566} C_DIS
LIN {X 0.246,Y -572.696,Z 1535.239,A 0.000,B 0.000,C 90.000,E1 78.926} C_DIS
LIN {X -0.002,Y -573.733,Z 1535.231,A 0.000,B 0.000,C 90.000,E1 77.589} C_DIS
LIN {X 0.214,Y -575.052,Z 1535.222,A 0.000,B 0.000,C 90.000,E1 75.936} C_DIS
LIN {X 0.258,Y -576.029,Z 1535.214,A 0.000,B 0.000,C 90.000,E1 74.574} C_DIS
LIN {X 0.111,Y -576.813,Z 1535.208,A 0.000,B 0.000,C 90.000,E1 73.504} C_DIS
LIN {X -0.191,Y -578.038,Z 1535.198,A 0.000,B 0.000,C 90.000,E1 71.638} C_DIS
LIN {X 0.269,Y -579.141,Z 1535.187,A 0.000,B 0.000,C 90.000,E1 69.699} C_DIS
LIN {X 0.142,Y -579.598,Z 1535.183,A 0.000,B 0.000,C 90.000,E1 68.901} C_DIS
LIN {X -0.246,Y -580.596,Z 1535.172,A 0.000,B 0.000,C 90.000,E1 67.050} C_DIS
LIN {X 0.113,Y -581.933,Z 1535.159,A 0.000,B 0.000,C 90.000,E1 64.588} C_DIS
LIN {X -0.279,Y -583.099,Z 1535.148,A 0.000,B 0.000,C 90.000,E1 62.743} C_DIS
LIN {X -0.132,Y -584.051,Z 1535.141,A 0.000,B 0.000,C 90.000,E1 61.385} C_DIS
LIN {X 0.054,Y -585.340,Z 1535.131,A 0.000,B 0.000,C 90.000,E1 59.488} C_DIS
LIN {X 0.319,Y -586.263,Z 1535.123,A 0.000,B 0.000,C 90.000,E1 58.122} C_DIS
LIN {X -0.068,Y -586.978,Z 1535.117,A 0.000,B 0.000,C 90.000,E1 57.089} C_DIS
LIN {X 0.105,Y -588.127,Z 1535.108,A 0.000,B 0.000,C 90.000,E1 55.468} C_DIS
LIN {X 0.276,Y -588.799,Z 1535.101,A 0.000,B 0.000,C 90.000,E1 54.116} C_DIS
LIN {X 0.262,Y -589.314,Z 1535.095,A 0.000,B 0.000,C 90.000,E1 53.050} C_DIS
LIN {X 0.249,Y -589.624,Z 1535.089,A 0.000,B 0.000,C 90.000,E1 51.984} C_DIS
LIN {X -0.081,Y -590.162,Z 1535.079,A 0.000,B 0.000,C 90.000,E1 50.150} C_DIS
LIN {X -0.179,Y -590.544,Z 1535.073,A 0.000,B 0.000,C 90.000,E1 49.094} C_DIS
LIN {X 0.363,Y -590.756,Z 1535.068,A 0.000,B 0.000,C 90.000,E1 48.243} C_DIS
LIN {X 0.076,Y -590.740,Z 1535.064,A 0.000,B 0.000,C 90.000,E1 47.472} C_DIS
LIN {X -0.214,Y -590.467,Z 1535.059,A 0.000,B 0.000,C 90.000,E1 46.701} C_DIS
LIN {X 0.140,Y -590.048,Z 1535.056,A 0.000,B 0.000,C 90.000,E1 46.134} C_DIS
LIN {X -0.341,Y -589.308,Z 1535.053,A 0.000,B 0.000,C 90.000,E1 45.648} C_DIS
LIN {X 0.009,Y -588.194,Z 1535.051,A 0.000,B 0.000,C 90.000,E1 45.081} C_DIS
LIN {X -0.235,Y -587.467,Z 1535.049,A 0.000,B 0.000,C 90.000,E1 44.838} C_DIS
LIN {X -0.069,Y -586.517,Z 1535.047,A 0.000,B 0.000,C 90.000,E1 44.555} C_DIS
LIN {X 0.101,Y -585.173,Z 1535.046,A 0.000,B 0.000,C 90.000,E1 44.271} C_DIS
LIN {X 0.321,Y -584.079,Z 1535.045,A 0.000,B 0.000,C 90.000,E1 44.109} C_DIS
LIN {X -0.365,Y -583.195,Z 1535.045,A 0.000,B 0.000,C 90.000,E1 44.109} C_DIS
LIN {X 0.161,Y -582.179,Z 1535.045,A 0.000,B 0.000,C 90.000,E1 44.028} C_DIS
LIN {X 0.091,Y -416.754,Z 1535.045,A 0.000,B 0.000,C 90.000,E1 44.028} C_DIS
LIN {X -0.077,Y -407.616,Z 1535.020,A 0.000,B 0.000,C 90.000,E1 39.564} C_DIS
LIN {X -0.204,Y -405.915,Z 1535.014,A 0.000,B 0.000,C 90.000,E1 38.543} C_DIS
LIN {X 0.013,Y -397.599,Z 1534.991,A 0.000,B 0.000,C 90.000,E1 34.326} C_DIS
LIN {X -0.121,Y -393.831,Z 1534.977,A 0.000,B 0.000,C 90.000,E1 31.878} C_DIS
LIN {X 0.000,Y -386.415,Z 1534.953,A 0.000,B 0.000,C 90.000,E1 27.590} C_DIS
LIN {X -0.016,Y -382.715,Z 1534.937,A 0.000,B 0.000,C 90.000,E1 24.719} C_DIS
LIN {X 0.075,Y -376.047,Z 1534.911,A 0.000,B 0.000,C 90.000,E1 19.993} C_DIS
LIN {X -0.065,Y -373.582,Z 1534.897,A 0.000,B 0.000,C 90.000,E1 17.457} C_DIS
LIN {X -0.031,Y -367.994,Z 1534.868,A 0.000,B 0.000,C 90.000,E1 12.299} C_DIS
LIN {X -0.014,Y -366.562,Z 1534.856,A 0.000,B 0.000,C 90.000,E1 10.074} C_DIS
LIN {X 0.059,Y -365.866,Z 1534.852,A 0.000,B 0.000,C 90.000,E1 9.321} C_DIS
LIN {X 0.073,Y -361.405,Z 1534.817,A 0.000,B 0.000,C 90.000,E1 2.980} C_DIS
LIN {X 0.164,Y -360.907,Z 1534.802,A 0.000,B 0.000,C 90.000,E1 0.344} C_DIS
LIN {X -0.058,Y -360.492,Z 1534.797,A 0.000,B 0.000,C 90.000,E1 359.427} C_DIS
LIN {X -0.053,Y -359.426,Z 1534.770,A 0.000,B 0.000,C 90.000,E1 354.546} C_DIS
LIN {X 0.070,Y -358.890,Z 1534.759,A 0.000,B 0.000,C 90.000,E1 352.648} C_DIS
LIN {X -0.020,Y -359.563,Z 1534.726,A 0.000,B 0.000,C 90.000,E1 346.645} C_DIS
LIN {X 0.001,Y -361.801,Z 1534.684,A 0.000,B 0.000,C 90.000,E1 339.135} C_DIS
LIN {X -0.154,Y -362.053,Z 1534.680,A 0.000,B 0.000,C 90.000,E1 338.411} C_DIS
LIN {X 0.189,Y -365.980,Z 1534.643,A 0.000,B 0.000,C 90.000,E1 331.641} C_DIS
LIN {X 0.029,Y -366.387,Z 1534.639,A 0.000,B 0.000,C 90.000,E1 330.923} C_DIS
LIN {X -0.031,Y -371.355,Z 1534.604,A 0.000,B 0.000,C 90.000,E1 324.642} C_DIS
LIN {X -0.043,Y -371.766,Z 1534.602,A 0.000,B 0.000,C 90.000,E1 324.276} C_DIS
LIN {X 0.013,Y -377.358,Z 1534.567,A 0.000,B 0.000,C 90.000,E1 318.038} C_DIS
LIN {X 0.012,Y -378.235,Z 1534.563,A 0.000,B 0.000,C 90.000,E1 317.310} C_DIS
LIN {X 0.002,Y -383.940,Z 1534.531,A 0.000,B 0.000,C 90.000,E1 311.515} C_DIS
LIN {X 0.088,Y -384.893,Z 1534.527,A 0.000,B 0.000,C 90.000,E1 310.782} C_DIS
LIN {X 0.262,Y -390.610,Z 1534.495,A 0.000,B 0.000,C 90.000,E1 305.025} C_DIS
LIN {X 0.106,Y -391.104,Z 1534.493,A 0.000,B 0.000,C 90.000,E1 304.692} C_DIS
LIN {X 0.022,Y -391.648,Z 1534.489,A 0.000,B 0.000,C 90.000,E1 303.992} C_DIS
LIN {X -0.080,Y -396.825,Z 1534.459,A 0.000,B 0.000,C 90.000,E1 298.693} C_DIS
LIN {X -0.210,Y -397.120,Z 1534.457,A 0.000,B 0.000,C 90.000,E1 298.359} C_DIS
LIN {X -0.055,Y -401.597,Z 1534.426,A 0.000,B 0.000,C 90.000,E1 292.717} C_DIS
LIN {X 0.222,Y -404.659,Z 1534.395,A 0.000,B 0.000,C 90.000,E1 287.094} C_DIS
LIN {X -0.079,Y -404.735,Z 1534.391,A 0.000,B 0.000,C 90.000,E1 286.441} C_DIS
LIN {X 0.214,Y -406.099,Z 1534.364,A 0.000,B 0.000,C 90.000,E1 281.535} C_DIS
LIN {X -0.176,Y -406.094,Z 1534.362,A 0.000,B 0.000,C 90.000,E1 281.243} C_DIS
LIN {X -0.097,Y -405.680,Z 1534.333,A 0.000,B 0.000,C 90.000,E1 276.024} C_DIS
LIN {X -0.165,Y -405.058,Z 1534.328,A 0.000,B 0.000,C 90.000,E1 274.992} C_DIS
LIN {X -0.060,Y -403.497,Z 1534.304,A 0.000,B 0.000,C 90.000,E1 270.802} C_DIS
LIN {X -0.092,Y -403.288,Z 1534.302,A 0.000,B 0.000,C 90.000,E1 270.458} C_DIS
LIN {X 0.091,Y -398.931,Z 1534.271,A 0.000,B 0.000,C 90.000,E1 264.837} C_DIS
LIN {X -0.040,Y -393.108,Z 1534.242,A 0.000,B 0.000,C 90.000,E1 259.567} C_DIS
LIN {X -0.079,Y -392.835,Z 1534.240,A 0.000,B 0.000,C 90.000,E1 259.218} C_DIS
LIN {X 0.034,Y -385.993,Z 1534.212,A 0.000,B 0.000,C 90.000,E1 254.212} C_DIS
LIN {X -0.026,Y -385.267,Z 1534.208,A 0.000,B 0.000,C 90.000,E1 253.504} C_DIS
LIN {X -0.004,Y -384.768,Z 1534.206,A 0.000,B 0.000,C 90.000,E1 253.142} C_DIS
LIN {X 0.221,Y -377.973,Z 1534.182,A 0.000,B 0.000,C 90.000,E1 248.773} C_DIS
LIN {X -0.044,Y -376.233,Z 1534.174,A 0.000,B 0.000,C 90.000,E1 247.358} C_DIS
LIN {X 0.057,Y -374.944,Z 1534.170,A 0.000,B 0.000,C 90.000,E1 246.613} C_DIS
LIN {X -0.208,Y -368.417,Z 1534.148,A 0.000,B 0.000,C 90.000,E1 242.615} C_DIS
LIN {X 0.097,Y -366.047,Z 1534.137,A 0.000,B 0.000,C 90.000,E1 240.717} C_DIS
LIN {X 0.004,Y -359.196,Z 1534.115,A 0.000,B 0.000,C 90.000,E1 236.628} C_DIS
LIN {X 0.021,Y -355.842,Z 1534.100,A 0.000,B 0.000,C 90.000,E1 233.989} C_DIS
LIN {X -0.173,Y -348.793,Z 1534.075,A 0.000,B 0.000,C 90.000,E1 229.461} C_DIS
LIN {X -0.097,Y -346.185,Z 1534.062,A 0.000,B 0.000,C 90.000,E1 227.148} C_DIS
LIN {X -0.088,Y -345.065,Z 1534.058,A 0.000,B 0.000,C 90.000,E1 226.377} C_DIS
LIN {X 0.094,Y -338.586,Z 1534.030,A 0.000,B 0.000,C 90.000,E1 221.310} C_DIS
LIN {X 0.094,Y -336.840,Z 1534.019,A 0.000,B 0.000,C 90.000,E1 219.358} C_DIS
LIN {X 0.014,Y -330.861,Z 1533.988,A 0.000,B 0.000,C 90.000,E1 213.865} C_DIS
LIN {X 0.149,Y -329.296,Z 1533.975,A 0.000,B 0.000,C 90.000,E1 211.465} C_DIS
LIN {X -0.154,Y -324.669,Z 1533.942,A 0.000,B 0.000,C 90.000,E1 205.540} C_DIS
LIN {X 0.174,Y -323.837,Z 1533.928,A 0.000,B 0.000,C 90.000,E1 203.078} C_DIS
LIN {X -0.017,Y -321.124,Z 1533.881,A 0.000,B 0.000,C 90.000,E1 194.662} C_DIS
LIN {X 0.138,Y -320.932,Z 1533.877,A 0.000,B 0.000,C 90.000,E1 193.828} C_DIS
LIN {X -0.076,Y -321.562,Z 1533.832,A 0.000,B 0.000,C 90.000,E1 185.796} C_DIS
LIN {X -0.143,Y -324.415,Z 1533.790,A 0.000,B 0.000,C 90.000,E1 178.165} C_DIS
LIN {X -0.141,Y -325.376,Z 1533.783,A 0.000,B 0.000,C 90.000,E1 176.963} C_DIS
LIN {X -0.100,Y -329.112,Z 1533.750,A 0.000,B 0.000,C 90.000,E1 170.971} C_DIS
LIN {X 0.061,Y -334.260,Z 1533.726,A 0.000,B 0.000,C 90.000,E1 166.589} C_DIS
LIN {X 0.067,Y -335.488,Z 1533.719,A 0.000,B 0.000,C 90.000,E1 165.408} C_DIS
LIN {X 0.143,Y -340.932,Z 1533.695,A 0.000,B 0.000,C 90.000,E1 161.094} C_DIS
LIN {X -0.172,Y -342.138,Z 1533.691,A 0.000,B 0.000,C 90.000,E1 160.369} C_DIS
LIN {X -0.058,Y -347.939,Z 1533.667,A 0.000,B 0.000,C 90.000,E1 156.102} C_DIS
LIN {X -0.081,Y -354.259,Z 1533.648,A 0.000,B 0.000,C 90.000,E1 152.666} C_DIS
LIN {X -0.222,Y -361.406,Z 1533.625,A 0.000,B 0.000,C 90.000,E1 148.535} C_DIS
LIN {X 0.065,Y -368.758,Z 1533.606,A 0.000,B 0.000,C 90.000,E1 145.135} C_DIS
LIN {X 0.065,Y -377.029,Z 1533.584,A 0.000,B 0.000,C 90.000,E1 141.090} C_DIS
LIN {X -0.061,Y -383.435,Z 1533.570,A 0.000,B 0.000,C 90.000,E1 138.566} C_DIS
LIN {X -0.015,Y -385.037,Z 1533.566,A 0.000,B 0.000,C 90.000,E1 137.838} C_DIS
LIN {X -0.004,Y -394.325,Z 1533.544,A 0.000,B 0.000,C 90.000,E1 133.905} C_DIS
LIN {X -0.038,Y -397.572,Z 1533.537,A 0.000,B 0.000,C 90.000,E1 132.732} C_DIS
LIN {X 0.308,Y -544.128,Z 1533.537,A 0.000,B 0.000,C 90.000,E1 132.690} C_DIS
LIN {X -0.023,Y -545.970,Z 1533.537,A 0.000,B 0.000,C 90.000,E1 132.609} C_DIS
LIN {X 0.048,Y -546.882,Z 1533.536,A 0.000,B 0.000,C 90.000,E1 132.486} C_DIS
LIN {X -0.156,Y -547.725,Z 1533.535,A 0.000,B 0.000,C 90.000,E1 132.366} C_DIS
LIN {X 0.042,Y -548.402,Z 1533.535,A 0.000,B 0.000,C 90.000,E1 132.204} C_DIS
LIN {X 0.079,Y -549.514,Z 1533.533,A 0.000,B 0.000,C 90.000,E1 131.919} C_DIS
LIN {X 0.118,Y -551.203,Z 1533.530,A 0.000,B 0.000,C 90.000,E1 131.353} C_DIS
LIN {X 0.221,Y -552.390,Z 1533.527,A 0.000,B 0.000,C 90.000,E1 130.782} C_DIS
LIN {X -0.018,Y -553.748,Z 1533.522,A 0.000,B 0.000,C 90.000,E1 129.967} C_DIS
LIN {X 0.111,Y -554.712,Z 1533.517,A 0.000,B 0.000,C 90.000,E1 129.116} C_DIS
LIN {X -0.034,Y -555.523,Z 1533.511,A 0.000,B 0.000,C 90.000,E1 128.016} C_DIS
LIN {X -0.019,Y -556.644,Z 1533.502,A 0.000,B 0.000,C 90.000,E1 126.343} C_DIS
LIN {X -0.027,Y -557.227,Z 1533.496,A 0.000,B 0.000,C 90.000,E1 125.231} C_DIS
LIN {X 0.057,Y -557.768,Z 1533.488,A 0.000,B 0.000,C 90.000,E1 123.833} C_DIS
LIN {X -0.238,Y -558.042,Z 1533.482,A 0.000,B 0.000,C 90.000,E1 122.752} C_DIS
LIN {X 0.097,Y -558.331,Z 1533.473,A 0.000,B 0.000,C 90.000,E1 121.052} C_DIS
LIN {X -0.136,Y -558.805,Z 1533.463,A 0.000,B 0.000,C 90.000,E1 119.411} C_DIS
LIN {X -0.065,Y -559.388,Z 1533.453,A 0.000,B 0.000,C 90.000,E1 117.462} C_DIS
LIN {X -0.033,Y -559.759,Z 1533.443,A 0.000,B 0.000,C 90.000,E1 115.796} C_DIS
LIN {X 0.301,Y -560.253,Z 1533.433,A 0.000,B 0.000,C 90.000,E1 113.823} C_DIS
LIN {X 0.183,Y -560.521,Z 1533.422,A 0.000,B 0.000,C 90.000,E1 111.897} C_DIS
LIN {X 0.177,Y -560.716,Z 1533.416,A 0.000,B 0.000,C 90.000,E1 110.791} C_DIS
LIN {X 0.198,Y -561.046,Z 1533.405,A 0.000,B 0.000,C 90.000,E1 108.852} C_DIS
LIN {X 0.226,Y -561.350,Z 1533.394,A 0.000,B 0.000,C 90.000,E1 106.913} C_DIS
LIN {X 0.318,Y -561.608,Z 1533.385,A 0.000,B 0.000,C 90.000,E1 105.245} C_DIS
LIN {X 0.035,Y -562.087,Z 1533.373,A 0.000,B 0.000,C 90.000,E1 103.063} C_DIS
LIN {X -0.198,Y -562.894,Z 1533.359,A 0.000,B 0.000,C 90.000,E1 100.602} C_DIS
LIN {X 0.263,Y -563.508,Z 1533.348,A 0.000,B 0.000,C 90.000,E1 98.624} C_DIS
LIN {X 0.018,Y -564.331,Z 1533.337,A 0.000,B 0.000,C 90.000,E1 96.720} C_DIS
LIN {X 0.202,Y -564.929,Z 1533.328,A 0.000,B 0.000,C 90.000,E1 95.049} C_DIS
LIN {X -0.105,Y -565.593,Z 1533.318,A 0.000,B 0.000,C 90.000,E1 93.154} C_DIS
LIN {X 0.165,Y -566.357,Z 1533.307,A 0.000,B 0.000,C 90.000,E1 91.203} C_DIS
LIN {X -0.266,Y -567.011,Z 1533.298,A 0.000,B 0.000,C 90.000,E1 89.599} C_DIS
LIN {X -0.241,Y -567.626,Z 1533.290,A 0.000,B 0.000,C 90.000,E1 88.224} C_DIS
LIN {X -0.043,Y -568.390,Z 1533.281,A 0.000,B 0.000,C 90.000,E1 86.560} C_DIS
LIN {X -0.271,Y -569.341,Z 1533.270,A 0.000,B 0.000,C 90.000,E1 84.666} C_DIS
LIN {X 0.013,Y -570.200,Z 1533.261,A 0.000,B 0.000,C 90.000,E1 82.996} C_DIS
LIN {X -0.180,Y -571.244,Z 1533.252,A 0.000,B 0.000,C 90.000,E1 81.376} C_DIS
LIN {X -0.231,Y -573.067,Z 1533.238,A 0.000,B 0.000,C 90.000,E1 78.926} C_DIS
LIN {X 0.211,Y -574.122,Z 1533.231,A 0.000,B 0.000,C 90.000,E1 77.521} C_DIS
LIN {X -0.249,Y -575.418,Z 1533.222,A 0.000,B 0.000,C 90.000,E1 75.936} C_DIS
LIN {X -0.201,Y -576.395,Z 1533.214,A 0.000,B 0.000,C 90.000,E1 74.574} C_DIS
LIN {X 0.210,Y -577.180,Z 1533.208,A 0.000,B 0.000,C 90.000,E1 73.449} C_DIS
LIN {X -0.088,Y -578.411,Z 1533.198,A 0.000,B 0.000,C 90.000,E1 71.583} C_DIS
LIN {X 0.189,Y -579.341,Z 1533.189,A 0.000,B 0.000,C 90.000,E1 69.934} C_DIS
LIN {X -0.291,Y -579.985,Z 1533.183,A 0.000,B 0.000,C 90.000,E1 68.901} C_DIS
LIN {X 0.091,Y -580.971,Z 1533.172,A 0.000,B 0.000,C 90.000,E1 66.975} C_DIS
LIN {X -0.170,Y -582.120,Z 1533.160,A 0.000,B 0.000,C 90.000,E1 64.845} C_DIS
LIN {X -0.037,Y -583.297,Z 1533.150,A 0.000,B 0.000,C 90.000,E1 62.948} C_DIS
LIN {X 0.260,Y -584.417,Z 1533.141,A 0.000,B 0.000,C 90.000,E1 61.307} C_DIS
LIN {X -0.040,Y -585.741,Z 1533.130,A 0.000,B 0.000,C 90.000,E1 59.459} C_DIS
LIN {X -0.067,Y -586.657,Z 1533.123,A 0.000,B 0.000,C 90.000,E1 58.122} C_DIS
LIN {X -0.088,Y -587.542,Z 1533.115,A 0.000,B 0.000,C 90.000,E1 56.786} C_DIS
LIN {X -0.269,Y -588.516,Z 1533.108,A 0.000,B 0.000,C 90.000,E1 55.468} C_DIS
LIN {X -0.092,Y -589.187,Z 1533.101,A 0.000,B 0.000,C 90.000,E1 54.116} C_DIS
LIN {X -0.101,Y -589.718,Z 1533.095,A 0.000,B 0.000,C 90.000,E1 53.050} C_DIS
LIN {X -0.108,Y -590.035,Z 1533.089,A 0.000,B 0.000,C 90.000,E1 51.984} C_DIS
LIN {X -0.049,Y -590.624,Z 1533.078,A 0.000,B 0.000,C 90.000,E1 50.114} C_DIS
LIN {X -0.132,Y -590.982,Z 1533.073,A 0.000,B 0.000,C 90.000,E1 49.057} C_DIS
LIN {X 0.027,Y -591.199,Z 1533.068,A 0.000,B 0.000,C 90.000,E1 48.243} C_DIS
LIN {X -0.061,Y -591.138,Z 1533.062,A 0.000,B 0.000,C 90.000,E1 47.187} C_DIS
LIN {X 0.056,Y -591.066,Z 1533.058,A 0.000,B 0.000,C 90.000,E1 46.377} C_DIS
LIN {X 0.004,Y -590.792,Z 1533.055,A 0.000,B 0.000,C 90.000,E1 45.850} C_DIS
LIN {X -0.299,Y -589.905,Z 1533.050,A 0.000,B 0.000,C 90.000,E1 45.081} C_DIS
LIN {X 0.054,Y -589.001,Z 1533.047,A 0.000,B 0.000,C 90.000,E1 44.514} C_DIS
LIN {X -0.188,Y -588.411,Z 1533.046,A 0.000,B 0.000,C 90.000,E1 44.271} C_DIS
LIN {X 0.400,Y -587.682,Z 1533.044,A 0.000,B 0.000,C 90.000,E1 43.947} C_DIS
LIN {X 0.154,Y -586.700,Z 1533.043,A 0.000,B 0.000,C 90.000,E1 43.704} C_DIS
LIN {X -0.095,Y -585.334,Z 1533.042,A 0.000,B 0.000,C 90.000,E1 43.461} C_DIS
LIN {X 0.191,Y -584.355,Z 1533.041,A 0.000,B 0.000,C 90.000,E1 43.299} C_DIS
LIN {X 0.077,Y -582.342,Z 1533.040,A 0.000,B 0.000,C 90.000,E1 43.176} C_DIS
LIN {X 0.047,Y -582.150,Z 1533.040,A 0.000,B 0.000,C 90.000,E1 43.176} C_DIS
LIN {X 0.012,Y -414.764,Z 1533.040,A 0.000,B 0.000,C 90.000,E1 43.176} C_DIS
LIN {X -0.018,Y -405.898,Z 1533.014,A 0.000,B 0.000,C 90.000,E1 38.508} C_DIS
LIN {X -0.053,Y -397.582,Z 1532.991,A 0.000,B 0.000,C 90.000,E1 34.326} C_DIS
LIN {X -0.187,Y -393.817,Z 1532.977,A 0.000,B 0.000,C 90.000,E1 31.878} C_DIS
LIN {X -0.065,Y -386.401,Z 1532.953,A 0.000,B 0.000,C 90.000,E1 27.590} C_DIS
LIN {X -0.082,Y -382.698,Z 1532.937,A 0.000,B 0.000,C 90.000,E1 24.719} C_DIS
LIN {X 0.009,Y -376.036,Z 1532.911,A 0.000,B 0.000,C 90.000,E1 19.993} C_DIS
LIN {X -0.130,Y -373.570,Z 1532.897,A 0.000,B 0.000,C 90.000,E1 17.457} C_DIS
LIN {X -0.096,Y -367.986,Z 1532.868,A 0.000,B 0.000,C 90.000,E1 12.299} C_DIS
LIN {X -0.078,Y -366.557,Z 1532.856,A 0.000,B 0.000,C 90.000,E1 10.074} C_DIS
LIN {X -0.005,Y -365.856,Z 1532.852,A 0.000,B 0.000,C 90.000,E1 9.321} C_DIS
LIN {X 0.009,Y -361.402,Z 1532.817,A 0.000,B 0.000,C 90.000,E1 2.980} C_DIS
LIN {X 0.100,Y -360.907,Z 1532.802,A 0.000,B 0.000,C 90.000,E1 0.344} C_DIS
LIN {X -0.058,Y -360.492,Z 1532.797,A 0.000,B 0.000,C 90.000,E1 359.427} C_DIS
LIN {X -0.053,Y -359.426,Z 1532.770,A 0.000,B 0.000,C 90.000,E1 354.546} C_DIS
LIN {X 0.070,Y -358.890,Z 1532.759,A 0.000,B 0.000,C 90.000,E1 352.648} C_DIS
LIN {X -0.020,Y -359.563,Z 1532.726,A 0.000,B 0.000,C 90.000,E1 346.645} C_DIS
LIN {X 0.001,Y -361.801,Z 1532.684,A 0.000,B 0.000,C 90.000,E1 339.135} C_DIS
LIN {X -0.154,Y -362.053,Z 1532.680,A 0.000,B 0.000,C 90.000,E1 338.411} C_DIS
LIN {X 0.189,Y -365.980,Z 1532.643,A 0.000,B 0.000,C 90.000,E1 331.641} C_DIS
LIN {X 0.029,Y -366.387,Z 1532.639,A 0.000,B 0.000,C 90.000,E1 330.923} C_DIS
LIN {X -0.031,Y -371.355,Z 1532.604,A 0.000,B 0.000,C 90.000,E1 324.642} C_DIS
LIN {X -0.043,Y -371.766,Z 1532.602,A 0.000,B 0.000,C 90.000,E1 324.276} C_DIS
LIN {X 0.013,Y -377.358,Z 1532.567,A 0.000,B 0.000,C 90.000,E1 318.038} C_DIS
LIN {X 0.012,Y -378.235,Z 1532.563,A 0.000,B 0.000,C 90.000,E1 317.310} C_DIS
LIN {X 0.002,Y -383.940,Z 1532.531,A 0.000,B 0.000,C 90.000,E1 311.515} C_DIS
LIN {X 0.088,Y -384.893,Z 1532.527,A 0.000,B 0.000,C 90.000,E1 310.782} C_DIS
LIN {X 0.262,Y -390.610,Z 1532.495,A 0.000,B 0.000,C 90.000,E1 305.025} C_DIS
LIN {X 0.106,Y -391.104,Z 1532.493,A 0.000,B 0.000,C 90.000,E1 304.692} C_DIS
LIN {X 0.022,Y -391.648,Z 1532.489,A 0.000,B 0.000,C 90.000,E1 303.992} C_DIS
LIN {X -0.080,Y -396.825,Z 1532.459,A 0.000,B 0.000,C 90.000,E1 298.693} C_DIS
LIN {X -0.210,Y -397.120,Z 1532.457,A 0.000,B 0.000,C 90.000,E1 298.359} C_DIS
LIN {X -0.055,Y -401.597,Z 1532.426,A 0.000,B 0.000,C 90.000,E1 292.717} C_DIS
LIN {X 0.222,Y -404.659,Z 1532.395,A 0.000,B 0.000,C 90.000,E1 287.094} C_DIS
LIN {X -0.079,Y -404.735,Z 1532.391,A 0.000,B 0.000,C 90.000,E1 286.441} C_DIS
LIN {X 0.214,Y -406.099,Z 1532.364,A 0.000,B 0.000,C 90.000,E1 281.535} C_DIS
LIN {X -0.176,Y -406.094,Z 1532.362,A 0.000,B 0.000,C 90.000,E1 281.243} C_DIS
LIN {X -0.097,Y -405.680,Z 1532.333,A 0.000,B 0.000,C 90.000,E1 276.024} C_DIS
LIN {X -0.165,Y -405.058,Z 1532.328,A 0.000,B 0.000,C 90.000,E1 274.992} C_DIS
LIN {X -0.060,Y -403.497,Z 1532.304,A 0.000,B 0.000,C 90.000,E1 270.802} C_DIS
LIN {X -0.092,Y -403.288,Z 1532.302,A 0.000,B 0.000,C 90.000,E1 270.458} C_DIS
LIN {X 0.091,Y -398.931,Z 1532.271,A 0.000,B 0.000,C 90.000,E1 264.837} C_DIS
LIN {X -0.040,Y -393.108,Z 1532.242,A 0.000,B 0.000,C 90.000,E1 259.567} C_DIS
LIN {X -0.079,Y -392.835,Z 1532.240,A 0.000,B 0.000,C 90.000,E1 259.218} C_DIS
LIN {X 0.034,Y -385.993,Z 1532.212,A 0.000,B 0.000,C 90.000,E1 254.212} C_DIS
LIN {X -0.026,Y -385.267,Z 1532.208,A 0.000,B 0.000,C 90.000,E1 253.504} C_DIS
LIN {X -0.004,Y -384.768,Z 1532.206,A 0.000,B 0.000,C 90.000,E1 253.142} C_DIS
LIN {X 0.221,Y -377.973,Z 1532.182,A 0.000,B 0.000,C 90.000,E1 248.773} C_DIS
LIN {X -0.044,Y -376.233,Z 1532.174,A 0.000,B 0.000,C 90.000,E1 247.358} C_DIS
LIN {X 0.057,Y -374.944,Z 1532.170,A 0.000,B 0.000,C 90.000,E1 246.613} C_DIS
LIN {X -0.208,Y -368.417,Z 1532.148,A 0.000,B 0.000,C 90.000,E1 242.615} C_DIS
LIN {X 0.097,Y -366.047,Z 1532.137,A 0.000,B 0.000,C 90.000,E1 240.717} C_DIS
LIN {X 0.004,Y -359.196,Z 1532.115,A 0.000,B 0.000,C 90.000,E1 236.628} C_DIS
LIN {X 0.021,Y -355.842,Z 1532.100,A 0.000,B 0.000,C 90.000,E1 233.989} C_DIS
LIN {X -0.173,Y -348.793,Z 1532.075,A 0.000,B 0.000,C 90.000,E1 229.461} C_DIS
LIN {X -0.097,Y -346.185,Z 1532.062,A 0.000,B 0.000,C 90.000,E1 227.148} C_DIS
LIN {X -0.088,Y -345.065,Z 1532.058,A 0.000,B 0.000,C 90.000,E1 226.377} C_DIS
LIN {X 0.094,Y -338.586,Z 1532.030,A 0.000,B 0.000,C 90.000,E1 221.310} C_DIS
LIN {X 0.094,Y -336.840,Z 1532.019,A 0.000,B 0.000,C 90.000,E1 219.358} C_DIS
LIN {X 0.014,Y -330.861,Z 1531.988,A 0.000,B 0.000,C 90.000,E1 213.865} C_DIS
LIN {X 0.149,Y -329.296,Z 1531.975,A 0.000,B 0.000,C 90.000,E1 211.465} C_DIS
LIN {X -0.154,Y -324.669,Z 1531.942,A 0.000,B 0.000,C 90.000,E1 205.540} C_DIS
LIN {X 0.174,Y -323.837,Z 1531.928,A 0.000,B 0.000,C 90.000,E1 203.078} C_DIS
LIN {X -0.017,Y -321.124,Z 1531.881,A 0.000,B 0.000,C 90.000,E1 194.662} C_DIS
LIN {X 0.138,Y -320.932,Z 1531.877,A 0.000,B 0.000,C 90.000,E1 193.828} C_DIS
LIN {X -0.076,Y -321.562,Z 1531.832,A 0.000,B 0.000,C 90.000,E1 185.796} C_DIS
LIN {X -0.143,Y -324.415,Z 1531.790,A 0.000,B 0.000,C 90.000,E1 178.165} C_DIS
LIN {X -0.141,Y -325.376,Z 1531.783,A 0.000,B 0.000,C 90.000,E1 176.963} C_DIS
LIN {X -0.100,Y -329.112,Z 1531.750,A 0.000,B 0.000,C 90.000,E1 170.971} C_DIS
LIN {X 0.061,Y -334.260,Z 1531.726,A 0.000,B 0.000,C 90.000,E1 166.589} C_DIS
LIN {X 0.067,Y -335.488,Z 1531.719,A 0.000,B 0.000,C 90.000,E1 165.408} C_DIS
LIN {X 0.143,Y -340.932,Z 1531.695,A 0.000,B 0.000,C 90.000,E1 161.094} C_DIS
LIN {X -0.172,Y -342.138,Z 1531.691,A 0.000,B 0.000,C 90.000,E1 160.369} C_DIS
LIN {X -0.058,Y -347.939,Z 1531.667,A 0.000,B 0.000,C 90.000,E1 156.102} C_DIS
LIN {X -0.081,Y -354.259,Z 1531.648,A 0.000,B 0.000,C 90.000,E1 152.666} C_DIS
LIN {X -0.222,Y -361.406,Z 1531.625,A 0.000,B 0.000,C 90.000,E1 148.535} C_DIS
LIN {X 0.065,Y -368.758,Z 1531.606,A 0.000,B 0.000,C 90.000,E1 145.135} C_DIS
LIN {X 0.065,Y -377.029,Z 1531.584,A 0.000,B 0.000,C 90.000,E1 141.090} C_DIS
LIN {X -0.061,Y -383.435,Z 1531.570,A 0.000,B 0.000,C 90.000,E1 138.566} C_DIS
LIN {X -0.015,Y -385.037,Z 1531.566,A 0.000,B 0.000,C 90.000,E1 137.838} C_DIS
LIN {X -0.135,Y -394.917,Z 1531.543,A 0.000,B 0.000,C 90.000,E1 133.704} C_DIS
LIN {X 0.013,Y -394.971,Z 1531.543,A 0.000,B 0.000,C 90.000,E1 133.662} C_DIS
LIN {X -0.029,Y -543.418,Z 1531.543,A 0.000,B 0.000,C 90.000,E1 133.662} C_DIS
LIN {X 0.298,Y -543.718,Z 1531.543,A 0.000,B 0.000,C 90.000,E1 133.623} C_DIS
LIN {X 0.084,Y -545.369,Z 1531.542,A 0.000,B 0.000,C 90.000,E1 133.542} C_DIS
LIN {X 0.128,Y -546.845,Z 1531.541,A 0.000,B 0.000,C 90.000,E1 133.338} C_DIS
LIN {X 0.127,Y -548.271,Z 1531.539,A 0.000,B 0.000,C 90.000,E1 133.056} C_DIS
LIN {X 0.159,Y -549.314,Z 1531.538,A 0.000,B 0.000,C 90.000,E1 132.771} C_DIS
LIN {X 0.202,Y -550.923,Z 1531.535,A 0.000,B 0.000,C 90.000,E1 132.204} C_DIS
LIN {X -0.114,Y -552.137,Z 1531.531,A 0.000,B 0.000,C 90.000,E1 131.676} C_DIS
LIN {X 0.360,Y -553.085,Z 1531.528,A 0.000,B 0.000,C 90.000,E1 131.067} C_DIS
LIN {X 0.125,Y -554.083,Z 1531.524,A 0.000,B 0.000,C 90.000,E1 130.253} C_DIS
LIN {X -0.024,Y -555.044,Z 1531.518,A 0.000,B 0.000,C 90.000,E1 129.152} C_DIS
LIN {X 0.263,Y -556.014,Z 1531.510,A 0.000,B 0.000,C 90.000,E1 127.729} C_DIS
LIN {X -0.202,Y -556.763,Z 1531.504,A 0.000,B 0.000,C 90.000,E1 126.664} C_DIS
LIN {X 0.206,Y -557.492,Z 1531.496,A 0.000,B 0.000,C 90.000,E1 125.231} C_DIS
LIN {X -0.015,Y -558.013,Z 1531.488,A 0.000,B 0.000,C 90.000,E1 123.865} C_DIS
LIN {X -0.078,Y -558.240,Z 1531.484,A 0.000,B 0.000,C 90.000,E1 123.038} C_DIS
LIN {X 0.054,Y -558.543,Z 1531.473,A 0.000,B 0.000,C 90.000,E1 121.082} C_DIS
LIN {X 0.115,Y -558.991,Z 1531.464,A 0.000,B 0.000,C 90.000,E1 119.411} C_DIS
LIN {X 0.191,Y -559.545,Z 1531.453,A 0.000,B 0.000,C 90.000,E1 117.462} C_DIS
LIN {X -0.278,Y -559.902,Z 1531.443,A 0.000,B 0.000,C 90.000,E1 115.848} C_DIS
LIN {X -0.175,Y -560.369,Z 1531.433,A 0.000,B 0.000,C 90.000,E1 113.898} C_DIS
LIN {X -0.073,Y -560.637,Z 1531.422,A 0.000,B 0.000,C 90.000,E1 111.950} C_DIS
LIN {X -0.081,Y -560.832,Z 1531.416,A 0.000,B 0.000,C 90.000,E1 110.844} C_DIS
LIN {X -0.062,Y -561.170,Z 1531.405,A 0.000,B 0.000,C 90.000,E1 108.906} C_DIS
LIN {X 0.195,Y -561.451,Z 1531.396,A 0.000,B 0.000,C 90.000,E1 107.221} C_DIS
LIN {X 0.054,Y -561.763,Z 1531.385,A 0.000,B 0.000,C 90.000,E1 105.300} C_DIS
LIN {X 0.161,Y -562.177,Z 1531.374,A 0.000,B 0.000,C 90.000,E1 103.355} C_DIS
LIN {X -0.071,Y -562.959,Z 1531.360,A 0.000,B 0.000,C 90.000,E1 100.894} C_DIS
LIN {X 0.236,Y -563.482,Z 1531.351,A 0.000,B 0.000,C 90.000,E1 99.208} C_DIS
LIN {X -0.089,Y -564.140,Z 1531.342,A 0.000,B 0.000,C 90.000,E1 97.587} C_DIS
LIN {X -0.092,Y -564.603,Z 1531.336,A 0.000,B 0.000,C 90.000,E1 96.486} C_DIS
LIN {X 0.041,Y -565.201,Z 1531.327,A 0.000,B 0.000,C 90.000,E1 94.821} C_DIS
LIN {X -0.224,Y -565.933,Z 1531.316,A 0.000,B 0.000,C 90.000,E1 92.922} C_DIS
LIN {X 0.026,Y -566.722,Z 1531.305,A 0.000,B 0.000,C 90.000,E1 90.974} C_DIS
LIN {X 0.171,Y -567.424,Z 1531.296,A 0.000,B 0.000,C 90.000,E1 89.312} C_DIS
LIN {X -0.224,Y -568.181,Z 1531.287,A 0.000,B 0.000,C 90.000,E1 87.707} C_DIS
LIN {X -0.042,Y -568.962,Z 1531.278,A 0.000,B 0.000,C 90.000,E1 86.045} C_DIS
LIN {X 0.237,Y -569.797,Z 1531.269,A 0.000,B 0.000,C 90.000,E1 84.375} C_DIS
LIN {X -0.028,Y -570.686,Z 1531.260,A 0.000,B 0.000,C 90.000,E1 82.761} C_DIS
LIN {X -0.203,Y -571.755,Z 1531.251,A 0.000,B 0.000,C 90.000,E1 81.141} C_DIS
LIN {X -0.065,Y -573.159,Z 1531.240,A 0.000,B 0.000,C 90.000,E1 79.218} C_DIS
LIN {X -0.103,Y -574.446,Z 1531.231,A 0.000,B 0.000,C 90.000,E1 77.589} C_DIS
LIN {X 0.128,Y -575.720,Z 1531.222,A 0.000,B 0.000,C 90.000,E1 75.936} C_DIS
LIN {X 0.183,Y -576.701,Z 1531.214,A 0.000,B 0.000,C 90.000,E1 74.574} C_DIS
LIN {X 0.046,Y -577.491,Z 1531.208,A 0.000,B 0.000,C 90.000,E1 73.504} C_DIS
LIN {X 0.142,Y -578.891,Z 1531.196,A 0.000,B 0.000,C 90.000,E1 71.329} C_DIS
LIN {X -0.272,Y -580.152,Z 1531.184,A 0.000,B 0.000,C 90.000,E1 69.209} C_DIS
LIN {X 0.253,Y -580.991,Z 1531.175,A 0.000,B 0.000,C 90.000,E1 67.539} C_DIS
LIN {X -0.134,Y -581.684,Z 1531.168,A 0.000,B 0.000,C 90.000,E1 66.230} C_DIS
LIN {X -0.138,Y -582.306,Z 1531.162,A 0.000,B 0.000,C 90.000,E1 65.153} C_DIS
LIN {X -0.120,Y -583.614,Z 1531.150,A 0.000,B 0.000,C 90.000,E1 62.999} C_DIS
LIN {X 0.036,Y -584.515,Z 1531.143,A 0.000,B 0.000,C 90.000,E1 61.641} C_DIS
LIN {X -0.181,Y -585.223,Z 1531.137,A 0.000,B 0.000,C 90.000,E1 60.589} C_DIS
LIN {X 0.115,Y -586.084,Z 1531.131,A 0.000,B 0.000,C 90.000,E1 59.488} C_DIS
LIN {X 0.265,Y -587.156,Z 1531.122,A 0.000,B 0.000,C 90.000,E1 57.867} C_DIS
LIN {X -0.114,Y -587.907,Z 1531.116,A 0.000,B 0.000,C 90.000,E1 56.834} C_DIS
LIN {X -0.082,Y -588.992,Z 1531.107,A 0.000,B 0.000,C 90.000,E1 55.229} C_DIS
LIN {X -0.028,Y -589.810,Z 1531.098,A 0.000,B 0.000,C 90.000,E1 53.623} C_DIS
LIN {X -0.237,Y -590.176,Z 1531.094,A 0.000,B 0.000,C 90.000,E1 52.844} C_DIS
LIN {X -0.293,Y -590.662,Z 1531.085,A 0.000,B 0.000,C 90.000,E1 51.251} C_DIS
LIN {X 0.027,Y -591.248,Z 1531.076,A 0.000,B 0.000,C 90.000,E1 49.622} C_DIS
LIN {X -0.297,Y -591.650,Z 1531.068,A 0.000,B 0.000,C 90.000,E1 48.324} C_DIS
LIN {X 0.021,Y -591.606,Z 1531.063,A 0.000,B 0.000,C 90.000,E1 47.229} C_DIS
LIN {X 0.339,Y -591.497,Z 1531.057,A 0.000,B 0.000,C 90.000,E1 46.134} C_DIS
LIN {X 0.051,Y -591.150,Z 1531.052,A 0.000,B 0.000,C 90.000,E1 45.364} C_DIS
LIN {X -0.007,Y -590.766,Z 1531.049,A 0.000,B 0.000,C 90.000,E1 44.838} C_DIS
LIN {X 0.352,Y -590.156,Z 1531.046,A 0.000,B 0.000,C 90.000,E1 44.271} C_DIS
LIN {X -0.128,Y -589.239,Z 1531.043,A 0.000,B 0.000,C 90.000,E1 43.785} C_DIS
LIN {X 0.217,Y -587.864,Z 1531.040,A 0.000,B 0.000,C 90.000,E1 43.218} C_DIS
LIN {X -0.030,Y -586.957,Z 1531.039,A 0.000,B 0.000,C 90.000,E1 42.975} C_DIS
LIN {X 0.150,Y -585.778,Z 1531.037,A 0.000,B 0.000,C 90.000,E1 42.690} C_DIS
LIN {X -0.388,Y -584.995,Z 1531.036,A 0.000,B 0.000,C 90.000,E1 42.609} C_DIS
LIN {X 0.017,Y -583.565,Z 1531.036,A 0.000,B 0.000,C 90.000,E1 42.405} C_DIS
LIN {X -0.117,Y -582.766,Z 1531.035,A 0.000,B 0.000,C 90.000,E1 42.366} C_DIS
LIN {X 0.094,Y -582.105,Z 1531.035,A 0.000,B 0.000,C 90.000,E1 42.324} C_DIS
LIN {X 0.031,Y -412.915,Z 1531.035,A 0.000,B 0.000,C 90.000,E1 42.324} C_DIS
LIN {X -0.041,Y -405.624,Z 1531.013,A 0.000,B 0.000,C 90.000,E1 38.382} C_DIS
LIN {X 0.020,Y -396.782,Z 1530.988,A 0.000,B 0.000,C 90.000,E1 33.833} C_DIS
LIN {X -0.005,Y -393.580,Z 1530.976,A 0.000,B 0.000,C 90.000,E1 31.720} C_DIS
LIN {X -0.098,Y -386.209,Z 1530.953,A 0.000,B 0.000,C 90.000,E1 27.462} C_DIS
LIN {X -0.119,Y -383.000,Z 1530.939,A 0.000,B 0.000,C 90.000,E1 24.951} C_DIS
LIN {X -0.162,Y -380.702,Z 1530.931,A 0.000,B 0.000,C 90.000,E1 23.515} C_DIS
LIN {X -0.120,Y -374.414,Z 1530.902,A 0.000,B 0.000,C 90.000,E1 18.417} C_DIS
LIN {X 0.164,Y -373.385,Z 1530.896,A 0.000,B 0.000,C 90.000,E1 17.275} C_DIS
LIN {X 0.180,Y -367.881,Z 1530.868,A 0.000,B 0.000,C 90.000,E1 12.119} C_DIS
LIN {X 0.124,Y -366.487,Z 1530.855,A 0.000,B 0.000,C 90.000,E1 9.905} C_DIS
LIN {X 0.059,Y -361.789,Z 1530.822,A 0.000,B 0.000,C 90.000,E1 3.955} C_DIS
LIN {X -0.055,Y -360.902,Z 1530.801,A 0.000,B 0.000,C 90.000,E1 0.229} C_DIS
LIN {X -0.053,Y -359.426,Z 1530.770,A 0.000,B 0.000,C 90.000,E1 354.546} C_DIS
LIN {X 0.070,Y -358.890,Z 1530.759,A 0.000,B 0.000,C 90.000,E1 352.648} C_DIS
LIN {X -0.020,Y -359.563,Z 1530.726,A 0.000,B 0.000,C 90.000,E1 346.645} C_DIS
LIN {X 0.001,Y -361.801,Z 1530.684,A 0.000,B 0.000,C 90.000,E1 339.135} C_DIS
LIN {X -0.154,Y -362.053,Z 1530.680,A 0.000,B 0.000,C 90.000,E1 338.411} C_DIS
LIN {X 0.189,Y -365.980,Z 1530.643,A 0.000,B 0.000,C 90.000,E1 331.641} C_DIS
LIN {X 0.029,Y -366.387,Z 1530.639,A 0.000,B 0.000,C 90.000,E1 330.923} C_DIS
LIN {X -0.031,Y -371.355,Z 1530.604,A 0.000,B 0.000,C 90.000,E1 324.642} C_DIS
LIN {X -0.043,Y -371.766,Z 1530.602,A 0.000,B 0.000,C 90.000,E1 324.276} C_DIS
LIN {X 0.013,Y -377.358,Z 1530.567,A 0.000,B 0.000,C 90.000,E1 318.038} C_DIS
LIN {X 0.012,Y -378.235,Z 1530.563,A 0.000,B 0.000,C 90.000,E1 317.310} C_DIS
LIN {X 0.002,Y -383.940,Z 1530.531,A 0.000,B 0.000,C 90.000,E1 311.515} C_DIS
LIN {X 0.088,Y -384.893,Z 1530.527,A 0.000,B 0.000,C 90.000,E1 310.782} C_DIS
LIN {X 0.262,Y -390.610,Z 1530.495,A 0.000,B 0.000,C 90.000,E1 305.025} C_DIS
LIN {X 0.106,Y -391.104,Z 1530.493,A 0.000,B 0.000,C 90.000,E1 304.692} C_DIS
LIN {X 0.022,Y -391.648,Z 1530.489,A 0.000,B 0.000,C 90.000,E1 303.992} C_DIS
LIN {X -0.080,Y -396.825,Z 1530.459,A 0.000,B 0.000,C 90.000,E1 298.693} C_DIS
LIN {X -0.210,Y -397.120,Z 1530.457,A 0.000,B 0.000,C 90.000,E1 298.359} C_DIS
LIN {X -0.055,Y -401.597,Z 1530.426,A 0.000,B 0.000,C 90.000,E1 292.717} C_DIS
LIN {X 0.222,Y -404.659,Z 1530.395,A 0.000,B 0.000,C 90.000,E1 287.094} C_DIS
LIN {X -0.079,Y -404.735,Z 1530.391,A 0.000,B 0.000,C 90.000,E1 286.441} C_DIS
LIN {X 0.214,Y -406.099,Z 1530.364,A 0.000,B 0.000,C 90.000,E1 281.535} C_DIS
LIN {X -0.176,Y -406.094,Z 1530.362,A 0.000,B 0.000,C 90.000,E1 281.243} C_DIS
LIN {X -0.097,Y -405.680,Z 1530.333,A 0.000,B 0.000,C 90.000,E1 276.024} C_DIS
LIN {X -0.165,Y -405.058,Z 1530.328,A 0.000,B 0.000,C 90.000,E1 274.992} C_DIS
LIN {X -0.060,Y -403.497,Z 1530.304,A 0.000,B 0.000,C 90.000,E1 270.802} C_DIS
LIN {X -0.092,Y -403.288,Z 1530.302,A 0.000,B 0.000,C 90.000,E1 270.458} C_DIS
LIN {X 0.091,Y -398.931,Z 1530.271,A 0.000,B 0.000,C 90.000,E1 264.837} C_DIS
LIN {X -0.040,Y -393.108,Z 1530.242,A 0.000,B 0.000,C 90.000,E1 259.567} C_DIS
LIN {X -0.079,Y -392.835,Z 1530.240,A 0.000,B 0.000,C 90.000,E1 259.218} C_DIS
LIN {X 0.034,Y -385.993,Z 1530.212,A 0.000,B 0.000,C 90.000,E1 254.212} C_DIS
LIN {X -0.026,Y -385.267,Z 1530.208,A 0.000,B 0.000,C 90.000,E1 253.504} C_DIS
LIN {X -0.004,Y -384.768,Z 1530.206,A 0.000,B 0.000,C 90.000,E1 253.142} C_DIS
LIN {X 0.221,Y -377.973,Z 1530.182,A 0.000,B 0.000,C 90.000,E1 248.773} C_DIS
LIN {X -0.044,Y -376.233,Z 1530.174,A 0.000,B 0.000,C 90.000,E1 247.358} C_DIS
LIN {X 0.057,Y -374.944,Z 1530.170,A 0.000,B 0.000,C 90.000,E1 246.613} C_DIS
LIN {X -0.208,Y -368.417,Z 1530.148,A 0.000,B 0.000,C 90.000,E1 242.615} C_DIS
LIN {X 0.097,Y -366.047,Z 1530.137,A 0.000,B 0.000,C 90.000,E1 240.717} C_DIS
LIN {X 0.004,Y -359.196,Z 1530.115,A 0.000,B 0.000,C 90.000,E1 236.628} C_DIS
LIN {X 0.021,Y -355.842,Z 1530.100,A 0.000,B 0.000,C 90.000,E1 233.989} C_DIS
LIN {X -0.173,Y -348.793,Z 1530.075,A 0.000,B 0.000,C 90.000,E1 229.461} C_DIS
LIN {X -0.097,Y -346.185,Z 1530.062,A 0.000,B 0.000,C 90.000,E1 227.148} C_DIS
LIN {X -0.088,Y -345.065,Z 1530.058,A 0.000,B 0.000,C 90.000,E1 226.377} C_DIS
LIN {X 0.094,Y -338.586,Z 1530.030,A 0.000,B 0.000,C 90.000,E1 221.310} C_DIS
LIN {X 0.094,Y -336.840,Z 1530.019,A 0.000,B 0.000,C 90.000,E1 219.358} C_DIS
LIN {X 0.014,Y -330.861,Z 1529.988,A 0.000,B 0.000,C 90.000,E1 213.865} C_DIS
LIN {X 0.149,Y -329.296,Z 1529.975,A 0.000,B 0.000,C 90.000,E1 211.465} C_DIS
LIN {X -0.154,Y -324.669,Z 1529.942,A 0.000,B 0.000,C 90.000,E1 205.540} C_DIS
LIN {X 0.174,Y -323.837,Z 1529.928,A 0.000,B 0.000,C 90.000,E1 203.078} C_DIS
LIN {X -0.017,Y -321.124,Z 1529.881,A 0.000,B 0.000,C 90.000,E1 194.662} C_DIS
LIN {X 0.138,Y -320.932,Z 1529.877,A 0.000,B 0.000,C 90.000,E1 193.828} C_DIS
LIN {X -0.076,Y -321.562,Z 1529.832,A 0.000,B 0.000,C 90.000,E1 185.796} C_DIS
LIN {X -0.143,Y -324.415,Z 1529.790,A 0.000,B 0.000,C 90.000,E1 178.165} C_DIS
LIN {X -0.141,Y -325.376,Z 1529.783,A 0.000,B 0.000,C 90.000,E1 176.963} C_DIS
LIN {X -0.100,Y -329.112,Z 1529.750,A 0.000,B 0.000,C 90.000,E1 170.971} C_DIS
LIN {X 0.061,Y -334.260,Z 1529.726,A 0.000,B 0.000,C 90.000,E1 166.589} C_DIS
LIN {X 0.067,Y -335.488,Z 1529.719,A 0.000,B 0.000,C 90.000,E1 165.408} C_DIS
LIN {X 0.143,Y -340.932,Z 1529.695,A 0.000,B 0.000,C 90.000,E1 161.094} C_DIS
LIN {X -0.172,Y -342.138,Z 1529.691,A 0.000,B 0.000,C 90.000,E1 160.369} C_DIS
LIN {X -0.058,Y -347.939,Z 1529.667,A 0.000,B 0.000,C 90.000,E1 156.102} C_DIS
LIN {X -0.081,Y -354.259,Z 1529.648,A 0.000,B 0.000,C 90.000,E1 152.666} C_DIS
LIN {X -0.222,Y -361.406,Z 1529.625,A 0.000,B 0.000,C 90.000,E1 148.535} C_DIS
LIN {X 0.065,Y -368.758,Z 1529.606,A 0.000,B 0.000,C 90.000,E1 145.135} C_DIS
LIN {X 0.065,Y -377.029,Z 1529.584,A 0.000,B 0.000,C 90.000,E1 141.090} C_DIS
LIN {X -0.061,Y -383.435,Z 1529.570,A 0.000,B 0.000,C 90.000,E1 138.566} C_DIS
LIN {X -0.015,Y -385.037,Z 1529.566,A 0.000,B 0.000,C 90.000,E1 137.838} C_DIS
LIN {X -0.129,Y -392.573,Z 1529.548,A 0.000,B 0.000,C 90.000,E1 134.595} C_DIS
LIN {X -0.235,Y -542.960,Z 1529.548,A 0.000,B 0.000,C 90.000,E1 134.595} C_DIS
LIN {X -0.171,Y -545.280,Z 1529.547,A 0.000,B 0.000,C 90.000,E1 134.433} C_DIS
LIN {X -0.106,Y -546.392,Z 1529.546,A 0.000,B 0.000,C 90.000,E1 134.271} C_DIS
LIN {X 0.292,Y -547.838,Z 1529.544,A 0.000,B 0.000,C 90.000,E1 133.947} C_DIS
LIN {X -0.078,Y -548.876,Z 1529.543,A 0.000,B 0.000,C 90.000,E1 133.704} C_DIS
LIN {X -0.036,Y -550.501,Z 1529.540,A 0.000,B 0.000,C 90.000,E1 133.137} C_DIS
LIN {X -0.358,Y -551.711,Z 1529.536,A 0.000,B 0.000,C 90.000,E1 132.609} C_DIS
LIN {X 0.112,Y -552.657,Z 1529.533,A 0.000,B 0.000,C 90.000,E1 132.000} C_DIS
LIN {X 0.236,Y -553.731,Z 1529.529,A 0.000,B 0.000,C 90.000,E1 131.148} C_DIS
LIN {X 0.145,Y -555.086,Z 1529.520,A 0.000,B 0.000,C 90.000,E1 129.483} C_DIS
LIN {X 0.082,Y -556.113,Z 1529.512,A 0.000,B 0.000,C 90.000,E1 128.096} C_DIS
LIN {X -0.046,Y -556.853,Z 1529.506,A 0.000,B 0.000,C 90.000,E1 126.996} C_DIS
LIN {X 0.032,Y -557.617,Z 1529.498,A 0.000,B 0.000,C 90.000,E1 125.598} C_DIS
LIN {X 0.047,Y -558.069,Z 1529.492,A 0.000,B 0.000,C 90.000,E1 124.485} C_DIS
LIN {X 0.149,Y -558.490,Z 1529.484,A 0.000,B 0.000,C 90.000,E1 123.086} C_DIS
LIN {X 0.063,Y -558.796,Z 1529.472,A 0.000,B 0.000,C 90.000,E1 120.875} C_DIS
LIN {X 0.124,Y -559.220,Z 1529.462,A 0.000,B 0.000,C 90.000,E1 119.205} C_DIS
LIN {X 0.199,Y -559.763,Z 1529.452,A 0.000,B 0.000,C 90.000,E1 117.257} C_DIS
LIN {X 0.232,Y -560.104,Z 1529.442,A 0.000,B 0.000,C 90.000,E1 115.591} C_DIS
LIN {X 0.029,Y -560.465,Z 1529.433,A 0.000,B 0.000,C 90.000,E1 113.951} C_DIS
LIN {X 0.126,Y -560.712,Z 1529.424,A 0.000,B 0.000,C 90.000,E1 112.280} C_DIS
LIN {X 0.128,Y -560.963,Z 1529.418,A 0.000,B 0.000,C 90.000,E1 111.173} C_DIS
LIN {X 0.132,Y -561.285,Z 1529.406,A 0.000,B 0.000,C 90.000,E1 108.960} C_DIS
LIN {X 0.081,Y -561.512,Z 1529.398,A 0.000,B 0.000,C 90.000,E1 107.583} C_DIS
LIN {X -0.053,Y -561.857,Z 1529.387,A 0.000,B 0.000,C 90.000,E1 105.662} C_DIS
LIN {X 0.064,Y -562.278,Z 1529.376,A 0.000,B 0.000,C 90.000,E1 103.716} C_DIS
LIN {X -0.041,Y -563.001,Z 1529.362,A 0.000,B 0.000,C 90.000,E1 101.243} C_DIS
LIN {X 0.265,Y -563.566,Z 1529.353,A 0.000,B 0.000,C 90.000,E1 99.557} C_DIS
LIN {X 0.102,Y -564.301,Z 1529.343,A 0.000,B 0.000,C 90.000,E1 97.644} C_DIS
LIN {X 0.192,Y -564.868,Z 1529.335,A 0.000,B 0.000,C 90.000,E1 96.258} C_DIS
LIN {X 0.235,Y -565.376,Z 1529.327,A 0.000,B 0.000,C 90.000,E1 94.878} C_DIS
LIN {X -0.169,Y -566.004,Z 1529.318,A 0.000,B 0.000,C 90.000,E1 93.269} C_DIS
LIN {X -0.138,Y -566.604,Z 1529.310,A 0.000,B 0.000,C 90.000,E1 91.892} C_DIS
LIN {X 0.018,Y -567.308,Z 1529.301,A 0.000,B 0.000,C 90.000,E1 90.229} C_DIS
LIN {X 0.053,Y -567.953,Z 1529.294,A 0.000,B 0.000,C 90.000,E1 88.854} C_DIS
LIN {X -0.214,Y -568.869,Z 1529.283,A 0.000,B 0.000,C 90.000,E1 86.963} C_DIS
LIN {X 0.177,Y -569.797,Z 1529.272,A 0.000,B 0.000,C 90.000,E1 85.008} C_DIS
LIN {X 0.029,Y -570.853,Z 1529.262,A 0.000,B 0.000,C 90.000,E1 83.109} C_DIS
LIN {X -0.226,Y -572.437,Z 1529.248,A 0.000,B 0.000,C 90.000,E1 80.679} C_DIS
LIN {X -0.079,Y -573.827,Z 1529.238,A 0.000,B 0.000,C 90.000,E1 78.757} C_DIS
LIN {X 0.165,Y -574.725,Z 1529.231,A 0.000,B 0.000,C 90.000,E1 77.645} C_DIS
LIN {X -0.153,Y -575.991,Z 1529.222,A 0.000,B 0.000,C 90.000,E1 76.047} C_DIS
LIN {X 0.120,Y -577.172,Z 1529.213,A 0.000,B 0.000,C 90.000,E1 74.393} C_DIS
LIN {X -0.010,Y -577.931,Z 1529.207,A 0.000,B 0.000,C 90.000,E1 73.323} C_DIS
LIN {X -0.284,Y -579.152,Z 1529.197,A 0.000,B 0.000,C 90.000,E1 71.456} C_DIS
LIN {X -0.185,Y -580.103,Z 1529.188,A 0.000,B 0.000,C 90.000,E1 69.826} C_DIS
LIN {X -0.059,Y -580.889,Z 1529.180,A 0.000,B 0.000,C 90.000,E1 68.465} C_DIS
LIN {X -0.050,Y -581.722,Z 1529.171,A 0.000,B 0.000,C 90.000,E1 66.847} C_DIS
LIN {X -0.025,Y -582.618,Z 1529.162,A 0.000,B 0.000,C 90.000,E1 65.229} C_DIS
LIN {X -0.009,Y -583.890,Z 1529.151,A 0.000,B 0.000,C 90.000,E1 63.076} C_DIS
LIN {X 0.147,Y -584.801,Z 1529.143,A 0.000,B 0.000,C 90.000,E1 61.719} C_DIS
LIN {X -0.071,Y -585.544,Z 1529.137,A 0.000,B 0.000,C 90.000,E1 60.667} C_DIS
LIN {X -0.107,Y -586.563,Z 1529.130,A 0.000,B 0.000,C 90.000,E1 59.331} C_DIS
LIN {X -0.121,Y -587.471,Z 1529.122,A 0.000,B 0.000,C 90.000,E1 57.995} C_DIS
LIN {X 0.190,Y -588.401,Z 1529.115,A 0.000,B 0.000,C 90.000,E1 56.628} C_DIS
LIN {X -0.105,Y -589.444,Z 1529.106,A 0.000,B 0.000,C 90.000,E1 55.055} C_DIS
LIN {X 0.294,Y -590.285,Z 1529.097,A 0.000,B 0.000,C 90.000,E1 53.417} C_DIS
LIN {X -0.173,Y -590.713,Z 1529.091,A 0.000,B 0.000,C 90.000,E1 52.396} C_DIS
LIN {X -0.049,Y -591.572,Z 1529.078,A 0.000,B 0.000,C 90.000,E1 49.989} C_DIS
LIN {X 0.117,Y -591.883,Z 1529.073,A 0.000,B 0.000,C 90.000,E1 49.175} C_DIS
LIN {X 0.040,Y -592.086,Z 1529.067,A 0.000,B 0.000,C 90.000,E1 48.119} C_DIS
LIN {X 0.121,Y -592.053,Z 1529.060,A 0.000,B 0.000,C 90.000,E1 46.782} C_DIS
LIN {X -0.351,Y -591.977,Z 1529.057,A 0.000,B 0.000,C 90.000,E1 46.296} C_DIS
LIN {X 0.147,Y -591.439,Z 1529.050,A 0.000,B 0.000,C 90.000,E1 44.919} C_DIS
LIN {X 0.274,Y -590.958,Z 1529.045,A 0.000,B 0.000,C 90.000,E1 44.109} C_DIS
LIN {X -0.202,Y -590.286,Z 1529.042,A 0.000,B 0.000,C 90.000,E1 43.623} C_DIS
LIN {X 0.149,Y -589.378,Z 1529.039,A 0.000,B 0.000,C 90.000,E1 43.056} C_DIS
LIN {X 0.093,Y -588.112,Z 1529.036,A 0.000,B 0.000,C 90.000,E1 42.528} C_DIS
LIN {X -0.155,Y -587.270,Z 1529.035,A 0.000,B 0.000,C 90.000,E1 42.285} C_DIS
LIN {X 0.032,Y -586.138,Z 1529.033,A 0.000,B 0.000,C 90.000,E1 42.000} C_DIS
LIN {X -0.220,Y -584.565,Z 1529.032,A 0.000,B 0.000,C 90.000,E1 41.757} C_DIS
LIN {X 0.009,Y -583.309,Z 1529.031,A 0.000,B 0.000,C 90.000,E1 41.595} C_DIS
LIN {X 0.142,Y -582.230,Z 1529.031,A 0.000,B 0.000,C 90.000,E1 41.515} C_DIS
LIN {X -0.026,Y -581.634,Z 1529.031,A 0.000,B 0.000,C 90.000,E1 41.515} C_DIS
LIN {X -0.043,Y -411.233,Z 1529.031,A 0.000,B 0.000,C 90.000,E1 41.515} C_DIS
LIN {X 0.021,Y -406.222,Z 1529.015,A 0.000,B 0.000,C 90.000,E1 38.705} C_DIS
LIN {X -0.151,Y -405.590,Z 1529.013,A 0.000,B 0.000,C 90.000,E1 38.382} C_DIS
LIN {X -0.088,Y -396.756,Z 1528.988,A 0.000,B 0.000,C 90.000,E1 33.833} C_DIS
LIN {X -0.113,Y -393.549,Z 1528.976,A 0.000,B 0.000,C 90.000,E1 31.720} C_DIS
LIN {X -0.027,Y -386.186,Z 1528.952,A 0.000,B 0.000,C 90.000,E1 27.436} C_DIS
LIN {X 0.121,Y -382.982,Z 1528.938,A 0.000,B 0.000,C 90.000,E1 24.899} C_DIS
LIN {X 0.113,Y -377.140,Z 1528.916,A 0.000,B 0.000,C 90.000,E1 20.918} C_DIS
LIN {X 0.083,Y -373.761,Z 1528.898,A 0.000,B 0.000,C 90.000,E1 17.638} C_DIS
LIN {X 0.031,Y -372.864,Z 1528.894,A 0.000,B 0.000,C 90.000,E1 16.913} C_DIS
LIN {X -0.067,Y -367.597,Z 1528.865,A 0.000,B 0.000,C 90.000,E1 11.771} C_DIS
LIN {X 0.018,Y -366.478,Z 1528.855,A 0.000,B 0.000,C 90.000,E1 9.905} C_DIS
LIN {X -0.045,Y -361.781,Z 1528.822,A 0.000,B 0.000,C 90.000,E1 3.955} C_DIS
LIN {X -0.160,Y -360.898,Z 1528.801,A 0.000,B 0.000,C 90.000,E1 0.229} C_DIS
LIN {X -0.053,Y -359.426,Z 1528.770,A 0.000,B 0.000,C 90.000,E1 354.546} C_DIS
LIN {X 0.070,Y -358.890,Z 1528.759,A 0.000,B 0.000,C 90.000,E1 352.648} C_DIS
LIN {X -0.020,Y -359.563,Z 1528.726,A 0.000,B 0.000,C 90.000,E1 346.645} C_DIS
LIN {X 0.001,Y -361.801,Z 1528.684,A 0.000,B 0.000,C 90.000,E1 339.135} C_DIS
LIN {X -0.154,Y -362.053,Z 1528.680,A 0.000,B 0.000,C 90.000,E1 338.411} C_DIS
LIN {X 0.189,Y -365.980,Z 1528.643,A 0.000,B 0.000,C 90.000,E1 331.641} C_DIS
LIN {X 0.029,Y -366.387,Z 1528.639,A 0.000,B 0.000,C 90.000,E1 330.923} C_DIS
LIN {X -0.031,Y -371.355,Z 1528.604,A 0.000,B 0.000,C 90.000,E1 324.642} C_DIS
LIN {X -0.043,Y -371.766,Z 1528.602,A 0.000,B 0.000,C 90.000,E1 324.276} C_DIS
LIN {X 0.013,Y -377.358,Z 1528.567,A 0.000,B 0.000,C 90.000,E1 318.038} C_DIS
LIN {X 0.012,Y -378.235,Z 1528.563,A 0.000,B 0.000,C 90.000,E1 317.310} C_DIS
LIN {X 0.002,Y -383.940,Z 1528.531,A 0.000,B 0.000,C 90.000,E1 311.515} C_DIS
LIN {X 0.088,Y -384.893,Z 1528.527,A 0.000,B 0.000,C 90.000,E1 310.782} C_DIS
LIN {X 0.262,Y -390.610,Z 1528.495,A 0.000,B 0.000,C 90.000,E1 305.025} C_DIS
LIN {X 0.106,Y -391.104,Z 1528.493,A 0.000,B 0.000,C 90.000,E1 304.692} C_DIS
LIN {X 0.022,Y -391.648,Z 1528.489,A 0.000,B 0.000,C 90.000,E1 303.992} C_DIS
LIN {X -0.080,Y -396.825,Z 1528.459,A 0.000,B 0.000,C 90.000,E1 298.693} C_DIS
LIN {X -0.210,Y -397.120,Z 1528.457,A 0.000,B 0.000,C 90.000,E1 298.359} C_DIS
LIN {X -0.055,Y -401.597,Z 1528.426,A 0.000,B 0.000,C 90.000,E1 292.717} C_DIS
LIN {X 0.222,Y -404.659,Z 1528.395,A 0.000,B 0.000,C 90.000,E1 287.094} C_DIS
LIN {X -0.079,Y -404.735,Z 1528.391,A 0.000,B 0.000,C 90.000,E1 286.441} C_DIS
LIN {X 0.214,Y -406.099,Z 1528.364,A 0.000,B 0.000,C 90.000,E1 281.535} C_DIS
LIN {X -0.176,Y -406.094,Z 1528.362,A 0.000,B 0.000,C 90.000,E1 281.243} C_DIS
LIN {X -0.097,Y -405.680,Z 1528.333,A 0.000,B 0.000,C 90.000,E1 276.024} C_DIS
LIN {X -0.165,Y -405.058,Z 1528.328,A 0.000,B 0.000,C 90.000,E1 274.992} C_DIS
LIN {X -0.060,Y -403.497,Z 1528.304,A 0.000,B 0.000,C 90.000,E1 270.802} C_DIS
LIN {X -0.092,Y -403.288,Z 1528.302,A 0.000,B 0.000,C 90.000,E1 270.458} C_DIS
LIN {X 0.091,Y -398.931,Z 1528.271,A 0.000,B 0.000,C 90.000,E1 264.837} C_DIS
LIN {X -0.040,Y -393.108,Z 1528.242,A 0.000,B 0.000,C 90.000,E1 259.567} C_DIS
LIN {X -0.079,Y -392.835,Z 1528.240,A 0.000,B 0.000,C 90.000,E1 259.218} C_DIS
LIN {X 0.034,Y -385.993,Z 1528.212,A 0.000,B 0.000,C 90.000,E1 254.212} C_DIS
LIN {X -0.026,Y -385.267,Z 1528.208,A 0.000,B 0.000,C 90.000,E1 253.504} C_DIS
LIN {X -0.004,Y -384.768,Z 1528.206,A 0.000,B 0.000,C 90.000,E1 253.142} C_DIS
LIN {X 0.221,Y -377.973,Z 1528.182,A 0.000,B 0.000,C 90.000,E1 248.773} C_DIS
LIN {X -0.044,Y -376.233,Z 1528.174,A 0.000,B 0.000,C 90.000,E1 247.358} C_DIS
LIN {X 0.057,Y -374.944,Z 1528.170,A 0.000,B 0.000,C 90.000,E1 246.613} C_DIS
LIN {X -0.208,Y -368.417,Z 1528.148,A 0.000,B 0.000,C 90.000,E1 242.615} C_DIS
LIN {X 0.097,Y -366.047,Z 1528.137,A 0.000,B 0.000,C 90.000,E1 240.717} C_DIS
LIN {X 0.004,Y -359.196,Z 1528.115,A 0.000,B 0.000,C 90.000,E1 236.628} C_DIS
LIN {X 0.021,Y -355.842,Z 1528.100,A 0.000,B 0.000,C 90.000,E1 233.989} C_DIS
LIN {X -0.173,Y -348.793,Z 1528.075,A 0.000,B 0.000,C 90.000,E1 229.461} C_DIS
LIN {X -0.097,Y -346.185,Z 1528.062,A 0.000,B 0.000,C 90.000,E1 227.148} C_DIS
LIN {X -0.088,Y -345.065,Z 1528.058,A 0.000,B 0.000,C 90.000,E1 226.377} C_DIS
LIN {X 0.094,Y -338.586,Z 1528.030,A 0.000,B 0.000,C 90.000,E1 221.310} C_DIS
LIN {X 0.094,Y -336.840,Z 1528.019,A 0.000,B 0.000,C 90.000,E1 219.358} C_DIS
LIN {X 0.014,Y -330.861,Z 1527.988,A 0.000,B 0.000,C 90.000,E1 213.865} C_DIS
LIN {X 0.149,Y -329.296,Z 1527.975,A 0.000,B 0.000,C 90.000,E1 211.465} C_DIS
LIN {X -0.154,Y -324.669,Z 1527.942,A 0.000,B 0.000,C 90.000,E1 205.540} C_DIS
LIN {X 0.174,Y -323.837,Z 1527.928,A 0.000,B 0.000,C 90.000,E1 203.078} C_DIS
LIN {X -0.017,Y -321.124,Z 1527.881,A 0.000,B 0.000,C 90.000,E1 194.662} C_DIS
LIN {X 0.138,Y -320.932,Z 1527.877,A 0.000,B 0.000,C 90.000,E1 193.828} C_DIS
LIN {X -0.076,Y -321.562,Z 1527.832,A 0.000,B 0.000,C 90.000,E1 185.796} C_DIS
LIN {X -0.143,Y -324.415,Z 1527.790,A 0.000,B 0.000,C 90.000,E1 178.165} C_DIS
LIN {X -0.141,Y -325.376,Z 1527.783,A 0.000,B 0.000,C 90.000,E1 176.963} C_DIS
LIN {X -0.100,Y -329.112,Z 1527.750,A 0.000,B 0.000,C 90.000,E1 170.971} C_DIS
LIN {X 0.061,Y -334.260,Z 1527.726,A 0.000,B 0.000,C 90.000,E1 166.589} C_DIS
LIN {X 0.067,Y -335.488,Z 1527.719,A 0.000,B 0.000,C 90.000,E1 165.408} C_DIS
LIN {X 0.143,Y -340.932,Z 1527.695,A 0.000,B 0.000,C 90.000,E1 161.094} C_DIS
LIN {X -0.172,Y -342.138,Z 1527.691,A 0.000,B 0.000,C 90.000,E1 160.369} C_DIS
LIN {X -0.058,Y -347.939,Z 1527.667,A 0.000,B 0.000,C 90.000,E1 156.102} C_DIS
LIN {X -0.081,Y -354.259,Z 1527.648,A 0.000,B 0.000,C 90.000,E1 152.666} C_DIS
LIN {X -0.222,Y -361.406,Z 1527.625,A 0.000,B 0.000,C 90.000,E1 148.535} C_DIS
LIN {X 0.065,Y -368.758,Z 1527.606,A 0.000,B 0.000,C 90.000,E1 145.135} C_DIS
LIN {X 0.065,Y -377.029,Z 1527.584,A 0.000,B 0.000,C 90.000,E1 141.090} C_DIS
LIN {X -0.061,Y -383.435,Z 1527.570,A 0.000,B 0.000,C 90.000,E1 138.566} C_DIS
LIN {X -0.015,Y -385.037,Z 1527.566,A 0.000,B 0.000,C 90.000,E1 137.838} C_DIS
LIN {X -0.102,Y -390.345,Z 1527.553,A 0.000,B 0.000,C 90.000,E1 135.486} C_DIS
LIN {X -0.188,Y -542.309,Z 1527.553,A 0.000,B 0.000,C 90.000,E1 135.486} C_DIS
LIN {X 0.030,Y -544.524,Z 1527.552,A 0.000,B 0.000,C 90.000,E1 135.324} C_DIS
LIN {X 0.065,Y -545.942,Z 1527.551,A 0.000,B 0.000,C 90.000,E1 135.121} C_DIS
LIN {X 0.073,Y -547.352,Z 1527.549,A 0.000,B 0.000,C 90.000,E1 134.838} C_DIS
LIN {X -0.297,Y -548.432,Z 1527.548,A 0.000,B 0.000,C 90.000,E1 134.595} C_DIS
LIN {X -0.256,Y -550.140,Z 1527.545,A 0.000,B 0.000,C 90.000,E1 134.028} C_DIS
LIN {X -0.203,Y -551.317,Z 1527.541,A 0.000,B 0.000,C 90.000,E1 133.461} C_DIS
LIN {X 0.261,Y -552.277,Z 1527.538,A 0.000,B 0.000,C 90.000,E1 132.852} C_DIS
LIN {X -0.028,Y -553.303,Z 1527.534,A 0.000,B 0.000,C 90.000,E1 132.043} C_DIS
LIN {X 0.159,Y -554.290,Z 1527.527,A 0.000,B 0.000,C 90.000,E1 130.906} C_DIS
LIN {X -0.278,Y -555.602,Z 1527.518,A 0.000,B 0.000,C 90.000,E1 129.277} C_DIS
LIN {X 0.012,Y -556.576,Z 1527.510,A 0.000,B 0.000,C 90.000,E1 127.855} C_DIS
LIN {X -0.003,Y -557.276,Z 1527.504,A 0.000,B 0.000,C 90.000,E1 126.744} C_DIS
LIN {X -0.038,Y -557.992,Z 1527.496,A 0.000,B 0.000,C 90.000,E1 125.358} C_DIS
LIN {X -0.108,Y -558.317,Z 1527.492,A 0.000,B 0.000,C 90.000,E1 124.532} C_DIS
LIN {X -0.315,Y -558.712,Z 1527.484,A 0.000,B 0.000,C 90.000,E1 123.166} C_DIS
LIN {X -0.101,Y -558.997,Z 1527.472,A 0.000,B 0.000,C 90.000,E1 120.924} C_DIS
LIN {X -0.317,Y -559.400,Z 1527.463,A 0.000,B 0.000,C 90.000,E1 119.283} C_DIS
LIN {X 0.026,Y -559.917,Z 1527.452,A 0.000,B 0.000,C 90.000,E1 117.308} C_DIS
LIN {X -0.188,Y -560.275,Z 1527.443,A 0.000,B 0.000,C 90.000,E1 115.668} C_DIS
LIN {X -0.152,Y -560.577,Z 1527.433,A 0.000,B 0.000,C 90.000,E1 114.003} C_DIS
LIN {X -0.059,Y -560.841,Z 1527.424,A 0.000,B 0.000,C 90.000,E1 112.333} C_DIS
LIN {X 0.254,Y -561.093,Z 1527.416,A 0.000,B 0.000,C 90.000,E1 110.918} C_DIS
LIN {X 0.162,Y -561.362,Z 1527.407,A 0.000,B 0.000,C 90.000,E1 109.268} C_DIS
LIN {X -0.113,Y -561.657,Z 1527.398,A 0.000,B 0.000,C 90.000,E1 107.638} C_DIS
LIN {X -0.101,Y -562.053,Z 1527.386,A 0.000,B 0.000,C 90.000,E1 105.426} C_DIS
LIN {X -0.134,Y -562.430,Z 1527.376,A 0.000,B 0.000,C 90.000,E1 103.772} C_DIS
LIN {X -0.238,Y -563.155,Z 1527.363,A 0.000,B 0.000,C 90.000,E1 101.299} C_DIS
LIN {X 0.067,Y -563.730,Z 1527.354,A 0.000,B 0.000,C 90.000,E1 99.613} C_DIS
LIN {X -0.095,Y -564.479,Z 1527.343,A 0.000,B 0.000,C 90.000,E1 97.701} C_DIS
LIN {X 0.092,Y -565.155,Z 1527.334,A 0.000,B 0.000,C 90.000,E1 96.030} C_DIS
LIN {X -0.268,Y -565.765,Z 1527.324,A 0.000,B 0.000,C 90.000,E1 94.416} C_DIS
LIN {X -0.104,Y -566.478,Z 1527.315,A 0.000,B 0.000,C 90.000,E1 92.751} C_DIS
LIN {X -0.074,Y -567.068,Z 1527.308,A 0.000,B 0.000,C 90.000,E1 91.375} C_DIS
LIN {X 0.199,Y -567.993,Z 1527.297,A 0.000,B 0.000,C 90.000,E1 89.427} C_DIS
LIN {X -0.062,Y -568.890,Z 1527.286,A 0.000,B 0.000,C 90.000,E1 87.535} C_DIS
LIN {X 0.012,Y -569.529,Z 1527.279,A 0.000,B 0.000,C 90.000,E1 86.159} C_DIS
LIN {X 0.134,Y -570.227,Z 1527.271,A 0.000,B 0.000,C 90.000,E1 84.780} C_DIS
LIN {X -0.124,Y -571.173,Z 1527.262,A 0.000,B 0.000,C 90.000,E1 83.166} C_DIS
LIN {X 0.005,Y -572.579,Z 1527.250,A 0.000,B 0.000,C 90.000,E1 80.971} C_DIS
LIN {X 0.155,Y -573.952,Z 1527.239,A 0.000,B 0.000,C 90.000,E1 79.050} C_DIS
LIN {X 0.248,Y -575.230,Z 1527.230,A 0.000,B 0.000,C 90.000,E1 77.409} C_DIS
LIN {X -0.057,Y -576.487,Z 1527.221,A 0.000,B 0.000,C 90.000,E1 75.811} C_DIS
LIN {X 0.225,Y -577.667,Z 1527.212,A 0.000,B 0.000,C 90.000,E1 74.157} C_DIS
LIN {X 0.099,Y -578.392,Z 1527.206,A 0.000,B 0.000,C 90.000,E1 73.087} C_DIS
LIN {X -0.168,Y -579.624,Z 1527.196,A 0.000,B 0.000,C 90.000,E1 71.221} C_DIS
LIN {X 0.135,Y -580.553,Z 1527.187,A 0.000,B 0.000,C 90.000,E1 69.571} C_DIS
LIN {X -0.121,Y -581.200,Z 1527.181,A 0.000,B 0.000,C 90.000,E1 68.518} C_DIS
LIN {X 0.070,Y -582.179,Z 1527.170,A 0.000,B 0.000,C 90.000,E1 66.613} C_DIS
LIN {X 0.338,Y -583.063,Z 1527.161,A 0.000,B 0.000,C 90.000,E1 64.973} C_DIS
LIN {X -0.027,Y -584.187,Z 1527.151,A 0.000,B 0.000,C 90.000,E1 63.127} C_DIS
LIN {X 0.142,Y -585.115,Z 1527.143,A 0.000,B 0.000,C 90.000,E1 61.769} C_DIS
LIN {X -0.190,Y -586.033,Z 1527.136,A 0.000,B 0.000,C 90.000,E1 60.461} C_DIS
LIN {X -0.092,Y -586.890,Z 1527.130,A 0.000,B 0.000,C 90.000,E1 59.380} C_DIS
LIN {X -0.219,Y -587.947,Z 1527.121,A 0.000,B 0.000,C 90.000,E1 57.788} C_DIS
LIN {X 0.104,Y -588.874,Z 1527.114,A 0.000,B 0.000,C 90.000,E1 56.421} C_DIS
LIN {X -0.048,Y -589.763,Z 1527.106,A 0.000,B 0.000,C 90.000,E1 55.102} C_DIS
LIN {X 0.224,Y -590.770,Z 1527.096,A 0.000,B 0.000,C 90.000,E1 53.210} C_DIS
LIN {X -0.030,Y -591.230,Z 1527.088,A 0.000,B 0.000,C 90.000,E1 51.904} C_DIS
LIN {X 0.062,Y -591.952,Z 1527.078,A 0.000,B 0.000,C 90.000,E1 50.033} C_DIS
LIN {X -0.001,Y -592.303,Z 1527.072,A 0.000,B 0.000,C 90.000,E1 48.976} C_DIS
LIN {X 0.174,Y -592.509,Z 1527.068,A 0.000,B 0.000,C 90.000,E1 48.162} C_DIS
LIN {X -0.133,Y -592.495,Z 1527.060,A 0.000,B 0.000,C 90.000,E1 46.863} C_DIS
LIN {X 0.000,Y -592.313,Z 1527.056,A 0.000,B 0.000,C 90.000,E1 46.053} C_DIS
LIN {X -0.098,Y -591.937,Z 1527.050,A 0.000,B 0.000,C 90.000,E1 45.000} C_DIS
LIN {X -0.201,Y -591.376,Z 1527.044,A 0.000,B 0.000,C 90.000,E1 43.947} C_DIS
LIN {X -0.079,Y -590.623,Z 1527.040,A 0.000,B 0.000,C 90.000,E1 43.137} C_DIS
LIN {X -0.128,Y -589.865,Z 1527.037,A 0.000,B 0.000,C 90.000,E1 42.609} C_DIS
LIN {X 0.066,Y -589.374,Z 1527.035,A 0.000,B 0.000,C 90.000,E1 42.324} C_DIS
LIN {X 0.408,Y -587.990,Z 1527.032,A 0.000,B 0.000,C 90.000,E1 41.757} C_DIS
LIN {X 0.159,Y -587.113,Z 1527.031,A 0.000,B 0.000,C 90.000,E1 41.515} C_DIS
LIN {X -0.093,Y -586.003,Z 1527.029,A 0.000,B 0.000,C 90.000,E1 41.272} C_DIS
LIN {X 0.092,Y -584.547,Z 1527.028,A 0.000,B 0.000,C 90.000,E1 40.987} C_DIS
LIN {X -0.009,Y -583.567,Z 1527.027,A 0.000,B 0.000,C 90.000,E1 40.862} C_DIS
LIN {X 0.271,Y -581.901,Z 1527.026,A 0.000,B 0.000,C 90.000,E1 40.701} C_DIS
LIN {X 0.036,Y -581.102,Z 1527.026,A 0.000,B 0.000,C 90.000,E1 40.701} C_DIS
LIN {X 0.002,Y -409.672,Z 1527.026,A 0.000,B 0.000,C 90.000,E1 40.701} C_DIS
LIN {X 0.042,Y -405.733,Z 1527.014,A 0.000,B 0.000,C 90.000,E1 38.418} C_DIS
LIN {X -0.071,Y -397.443,Z 1526.990,A 0.000,B 0.000,C 90.000,E1 34.246} C_DIS
LIN {X 0.121,Y -393.678,Z 1526.977,A 0.000,B 0.000,C 90.000,E1 31.750} C_DIS
LIN {X -0.110,Y -386.279,Z 1526.953,A 0.000,B 0.000,C 90.000,E1 27.513} C_DIS
LIN {X 0.049,Y -383.055,Z 1526.939,A 0.000,B 0.000,C 90.000,E1 24.975} C_DIS
LIN {X 0.018,Y -381.945,Z 1526.935,A 0.000,B 0.000,C 90.000,E1 24.259} C_DIS
LIN {X -0.213,Y -375.548,Z 1526.909,A 0.000,B 0.000,C 90.000,E1 19.577} C_DIS
LIN {X 0.024,Y -373.454,Z 1526.896,A 0.000,B 0.000,C 90.000,E1 17.347} C_DIS
LIN {X 0.068,Y -367.920,Z 1526.868,A 0.000,B 0.000,C 90.000,E1 12.187} C_DIS
LIN {X 0.088,Y -366.513,Z 1526.855,A 0.000,B 0.000,C 90.000,E1 9.962} C_DIS
LIN {X 0.023,Y -361.811,Z 1526.822,A 0.000,B 0.000,C 90.000,E1 4.012} C_DIS
LIN {X -0.092,Y -360.904,Z 1526.802,A 0.000,B 0.000,C 90.000,E1 0.286} C_DIS
LIN {X -0.053,Y -359.426,Z 1526.770,A 0.000,B 0.000,C 90.000,E1 354.546} C_DIS
LIN {X 0.070,Y -358.890,Z 1526.759,A 0.000,B 0.000,C 90.000,E1 352.648} C_DIS
LIN {X -0.020,Y -359.563,Z 1526.726,A 0.000,B 0.000,C 90.000,E1 346.645} C_DIS
LIN {X 0.001,Y -361.801,Z 1526.684,A 0.000,B 0.000,C 90.000,E1 339.135} C_DIS
LIN {X -0.154,Y -362.053,Z 1526.680,A 0.000,B 0.000,C 90.000,E1 338.411} C_DIS
LIN {X 0.189,Y -365.980,Z 1526.643,A 0.000,B 0.000,C 90.000,E1 331.641} C_DIS
LIN {X 0.029,Y -366.387,Z 1526.639,A 0.000,B 0.000,C 90.000,E1 330.923} C_DIS
LIN {X -0.031,Y -371.355,Z 1526.604,A 0.000,B 0.000,C 90.000,E1 324.642} C_DIS
LIN {X -0.043,Y -371.766,Z 1526.602,A 0.000,B 0.000,C 90.000,E1 324.276} C_DIS
LIN {X 0.013,Y -377.358,Z 1526.567,A 0.000,B 0.000,C 90.000,E1 318.038} C_DIS
LIN {X 0.012,Y -378.235,Z 1526.563,A 0.000,B 0.000,C 90.000,E1 317.310} C_DIS
LIN {X 0.002,Y -383.940,Z 1526.531,A 0.000,B 0.000,C 90.000,E1 311.515} C_DIS
LIN {X 0.088,Y -384.893,Z 1526.527,A 0.000,B 0.000,C 90.000,E1 310.782} C_DIS
LIN {X 0.262,Y -390.610,Z 1526.495,A 0.000,B 0.000,C 90.000,E1 305.025} C_DIS
LIN {X 0.106,Y -391.104,Z 1526.493,A 0.000,B 0.000,C 90.000,E1 304.692} C_DIS
LIN {X 0.022,Y -391.648,Z 1526.489,A 0.000,B 0.000,C 90.000,E1 303.992} C_DIS
LIN {X -0.080,Y -396.825,Z 1526.459,A 0.000,B 0.000,C 90.000,E1 298.693} C_DIS
LIN {X -0.210,Y -397.120,Z 1526.457,A 0.000,B 0.000,C 90.000,E1 298.359} C_DIS
LIN {X -0.055,Y -401.597,Z 1526.426,A 0.000,B 0.000,C 90.000,E1 292.717} C_DIS
LIN {X 0.222,Y -404.659,Z 1526.395,A 0.000,B 0.000,C 90.000,E1 287.094} C_DIS
LIN {X -0.079,Y -404.735,Z 1526.391,A 0.000,B 0.000,C 90.000,E1 286.441} C_DIS
LIN {X 0.214,Y -406.099,Z 1526.364,A 0.000,B 0.000,C 90.000,E1 281.535} C_DIS
LIN {X -0.176,Y -406.094,Z 1526.362,A 0.000,B 0.000,C 90.000,E1 281.243} C_DIS
LIN {X -0.097,Y -405.680,Z 1526.333,A 0.000,B 0.000,C 90.000,E1 276.024} C_DIS
LIN {X -0.165,Y -405.058,Z 1526.328,A 0.000,B 0.000,C 90.000,E1 274.992} C_DIS
LIN {X -0.060,Y -403.497,Z 1526.304,A 0.000,B 0.000,C 90.000,E1 270.802} C_DIS
LIN {X -0.092,Y -403.288,Z 1526.302,A 0.000,B 0.000,C 90.000,E1 270.458} C_DIS
LIN {X 0.091,Y -398.931,Z 1526.271,A 0.000,B 0.000,C 90.000,E1 264.837} C_DIS
LIN {X -0.040,Y -393.108,Z 1526.242,A 0.000,B 0.000,C 90.000,E1 259.567} C_DIS
LIN {X -0.079,Y -392.835,Z 1526.240,A 0.000,B 0.000,C 90.000,E1 259.218} C_DIS
LIN {X 0.034,Y -385.993,Z 1526.212,A 0.000,B 0.000,C 90.000,E1 254.212} C_DIS
LIN {X -0.026,Y -385.267,Z 1526.208,A 0.000,B 0.000,C 90.000,E1 253.504} C_DIS
LIN {X -0.004,Y -384.768,Z 1526.206,A 0.000,B 0.000,C 90.000,E1 253.142} C_DIS
LIN {X 0.221,Y -377.973,Z 1526.182,A 0.000,B 0.000,C 90.000,E1 248.773} C_DIS
LIN {X -0.044,Y -376.233,Z 1526.174,A 0.000,B 0.000,C 90.000,E1 247.358} C_DIS
LIN {X 0.057,Y -374.944,Z 1526.170,A 0.000,B 0.000,C 90.000,E1 246.613} C_DIS
LIN {X -0.208,Y -368.417,Z 1526.148,A 0.000,B 0.000,C 90.000,E1 242.615} C_DIS
LIN {X 0.097,Y -366.047,Z 1526.137,A 0.000,B 0.000,C 90.000,E1 240.717} C_DIS
LIN {X 0.004,Y -359.196,Z 1526.115,A 0.000,B 0.000,C 90.000,E1 236.628} C_DIS
LIN {X 0.021,Y -355.842,Z 1526.100,A 0.000,B 0.000,C 90.000,E1 233.989} C_DIS
LIN {X -0.173,Y -348.793,Z 1526.075,A 0.000,B 0.000,C 90.000,E1 229.461} C_DIS
LIN {X -0.097,Y -346.185,Z 1526.062,A 0.000,B 0.000,C 90.000,E1 227.148} C_DIS
LIN {X -0.088,Y -345.065,Z 1526.058,A 0.000,B 0.000,C 90.000,E1 226.377} C_DIS
LIN {X 0.094,Y -338.586,Z 1526.030,A 0.000,B 0.000,C 90.000,E1 221.310} C_DIS
LIN {X 0.094,Y -336.840,Z 1526.019,A 0.000,B 0.000,C 90.000,E1 219.358} C_DIS
LIN {X 0.014,Y -330.861,Z 1525.988,A 0.000,B 0.000,C 90.000,E1 213.865} C_DIS
LIN {X 0.149,Y -329.296,Z 1525.975,A 0.000,B 0.000,C 90.000,E1 211.465} C_DIS
LIN {X -0.154,Y -324.669,Z 1525.942,A 0.000,B 0.000,C 90.000,E1 205.540} C_DIS
LIN {X 0.174,Y -323.837,Z 1525.928,A 0.000,B 0.000,C 90.000,E1 203.078} C_DIS
LIN {X -0.017,Y -321.124,Z 1525.881,A 0.000,B 0.000,C 90.000,E1 194.662} C_DIS
LIN {X 0.138,Y -320.932,Z 1525.877,A 0.000,B 0.000,C 90.000,E1 193.828} C_DIS
LIN {X -0.076,Y -321.562,Z 1525.832,A 0.000,B 0.000,C 90.000,E1 185.796} C_DIS
LIN {X -0.143,Y -324.415,Z 1525.790,A 0.000,B 0.000,C 90.000,E1 178.165} C_DIS
LIN {X -0.141,Y -325.376,Z 1525.783,A 0.000,B 0.000,C 90.000,E1 176.963} C_DIS
LIN {X -0.100,Y -329.112,Z 1525.750,A 0.000,B 0.000,C 90.000,E1 170.971} C_DIS
LIN {X 0.061,Y -334.260,Z 1525.726,A 0.000,B 0.000,C 90.000,E1 166.589} C_DIS
LIN {X 0.067,Y -335.488,Z 1525.719,A 0.000,B 0.000,C 90.000,E1 165.408} C_DIS
LIN {X 0.143,Y -340.932,Z 1525.695,A 0.000,B 0.000,C 90.000,E1 161.094} C_DIS
LIN {X -0.172,Y -342.138,Z 1525.691,A 0.000,B 0.000,C 90.000,E1 160.369} C_DIS
LIN {X -0.058,Y -347.939,Z 1525.667,A 0.000,B 0.000,C 90.000,E1 156.102} C_DIS
LIN {X -0.081,Y -354.259,Z 1525.648,A 0.000,B 0.000,C 90.000,E1 152.666} C_DIS
LIN {X -0.222,Y -361.406,Z 1525.625,A 0.000,B 0.000,C 90.000,E1 148.535} C_DIS
LIN {X 0.065,Y -368.758,Z 1525.606,A 0.000,B 0.000,C 90.000,E1 145.135} C_DIS
LIN {X 0.065,Y -377.029,Z 1525.584,A 0.000,B 0.000,C 90.000,E1 141.090} C_DIS
LIN {X -0.061,Y -383.435,Z 1525.570,A 0.000,B 0.000,C 90.000,E1 138.566} C_DIS
LIN {X -0.015,Y -385.037,Z 1525.566,A 0.000,B 0.000,C 90.000,E1 137.838} C_DIS
LIN {X -0.216,Y -388.287,Z 1525.557,A 0.000,B 0.000,C 90.000,E1 136.377} C_DIS
LIN {X 0.025,Y -541.696,Z 1525.557,A 0.000,B 0.000,C 90.000,E1 136.338} C_DIS
LIN {X -0.022,Y -541.914,Z 1525.557,A 0.000,B 0.000,C 90.000,E1 136.338} C_DIS
LIN {X -0.255,Y -543.980,Z 1525.557,A 0.000,B 0.000,C 90.000,E1 136.215} C_DIS
LIN {X -0.112,Y -545.076,Z 1525.556,A 0.000,B 0.000,C 90.000,E1 136.053} C_DIS
LIN {X 0.280,Y -546.602,Z 1525.554,A 0.000,B 0.000,C 90.000,E1 135.729} C_DIS
LIN {X -0.092,Y -547.740,Z 1525.553,A 0.000,B 0.000,C 90.000,E1 135.486} C_DIS
LIN {X -0.074,Y -548.671,Z 1525.551,A 0.000,B 0.000,C 90.000,E1 135.202} C_DIS
LIN {X -0.034,Y -550.152,Z 1525.548,A 0.000,B 0.000,C 90.000,E1 134.636} C_DIS
LIN {X -0.365,Y -551.323,Z 1525.545,A 0.000,B 0.000,C 90.000,E1 134.109} C_DIS
LIN {X 0.097,Y -552.168,Z 1525.542,A 0.000,B 0.000,C 90.000,E1 133.500} C_DIS
LIN {X -0.186,Y -553.096,Z 1525.537,A 0.000,B 0.000,C 90.000,E1 132.690} C_DIS
LIN {X 0.016,Y -554.350,Z 1525.529,A 0.000,B 0.000,C 90.000,E1 131.272} C_DIS
LIN {X -0.071,Y -555.453,Z 1525.522,A 0.000,B 0.000,C 90.000,E1 129.886} C_DIS
LIN {X 0.227,Y -556.431,Z 1525.514,A 0.000,B 0.000,C 90.000,E1 128.463} C_DIS
LIN {X 0.187,Y -557.342,Z 1525.506,A 0.000,B 0.000,C 90.000,E1 127.076} C_DIS
LIN {X -0.176,Y -558.086,Z 1525.498,A 0.000,B 0.000,C 90.000,E1 125.724} C_DIS
LIN {X -0.159,Y -558.532,Z 1525.492,A 0.000,B 0.000,C 90.000,E1 124.612} C_DIS
LIN {X -0.053,Y -558.919,Z 1525.484,A 0.000,B 0.000,C 90.000,E1 123.214} C_DIS
LIN {X 0.081,Y -559.089,Z 1525.474,A 0.000,B 0.000,C 90.000,E1 121.258} C_DIS
LIN {X -0.065,Y -559.525,Z 1525.463,A 0.000,B 0.000,C 90.000,E1 119.333} C_DIS
LIN {X 0.014,Y -560.022,Z 1525.452,A 0.000,B 0.000,C 90.000,E1 117.385} C_DIS
LIN {X 0.053,Y -560.378,Z 1525.443,A 0.000,B 0.000,C 90.000,E1 115.720} C_DIS
LIN {X 0.166,Y -560.721,Z 1525.432,A 0.000,B 0.000,C 90.000,E1 113.770} C_DIS
LIN {X -0.247,Y -560.976,Z 1525.423,A 0.000,B 0.000,C 90.000,E1 112.153} C_DIS
LIN {X -0.243,Y -561.209,Z 1525.417,A 0.000,B 0.000,C 90.000,E1 111.046} C_DIS
LIN {X -0.017,Y -561.513,Z 1525.406,A 0.000,B 0.000,C 90.000,E1 109.087} C_DIS
LIN {X 0.248,Y -561.797,Z 1525.397,A 0.000,B 0.000,C 90.000,E1 107.402} C_DIS
LIN {X 0.120,Y -562.175,Z 1525.386,A 0.000,B 0.000,C 90.000,E1 105.481} C_DIS
LIN {X 0.242,Y -562.613,Z 1525.375,A 0.000,B 0.000,C 90.000,E1 103.536} C_DIS
LIN {X 0.031,Y -563.375,Z 1525.362,A 0.000,B 0.000,C 90.000,E1 101.074} C_DIS
LIN {X -0.041,Y -564.078,Z 1525.351,A 0.000,B 0.000,C 90.000,E1 99.151} C_DIS
LIN {X 0.210,Y -564.749,Z 1525.342,A 0.000,B 0.000,C 90.000,E1 97.473} C_DIS
LIN {X -0.093,Y -565.428,Z 1525.333,A 0.000,B 0.000,C 90.000,E1 95.853} C_DIS
LIN {X 0.210,Y -566.209,Z 1525.322,A 0.000,B 0.000,C 90.000,E1 93.898} C_DIS
LIN {X -0.097,Y -567.048,Z 1525.311,A 0.000,B 0.000,C 90.000,E1 92.007} C_DIS
LIN {X 0.067,Y -567.799,Z 1525.302,A 0.000,B 0.000,C 90.000,E1 90.344} C_DIS
LIN {X 0.112,Y -568.468,Z 1525.294,A 0.000,B 0.000,C 90.000,E1 88.969} C_DIS
LIN {X -0.142,Y -569.438,Z 1525.284,A 0.000,B 0.000,C 90.000,E1 87.078} C_DIS
LIN {X 0.266,Y -570.386,Z 1525.273,A 0.000,B 0.000,C 90.000,E1 85.122} C_DIS
LIN {X -0.044,Y -571.294,Z 1525.264,A 0.000,B 0.000,C 90.000,E1 83.514} C_DIS
LIN {X -0.213,Y -572.316,Z 1525.255,A 0.000,B 0.000,C 90.000,E1 81.894} C_DIS
LIN {X 0.206,Y -573.442,Z 1525.246,A 0.000,B 0.000,C 90.000,E1 80.218} C_DIS
LIN {X 0.282,Y -574.615,Z 1525.237,A 0.000,B 0.000,C 90.000,E1 78.578} C_DIS
LIN {X 0.188,Y -575.706,Z 1525.229,A 0.000,B 0.000,C 90.000,E1 77.229} C_DIS
LIN {X -0.245,Y -576.972,Z 1525.220,A 0.000,B 0.000,C 90.000,E1 75.644} C_DIS
LIN {X -0.174,Y -577.916,Z 1525.213,A 0.000,B 0.000,C 90.000,E1 74.283} C_DIS
LIN {X 0.072,Y -578.826,Z 1525.205,A 0.000,B 0.000,C 90.000,E1 72.906} C_DIS
LIN {X 0.203,Y -580.243,Z 1525.193,A 0.000,B 0.000,C 90.000,E1 70.732} C_DIS
LIN {X 0.021,Y -581.465,Z 1525.181,A 0.000,B 0.000,C 90.000,E1 68.592} C_DIS
LIN {X -0.326,Y -582.464,Z 1525.171,A 0.000,B 0.000,C 90.000,E1 66.741} C_DIS
LIN {X -0.183,Y -583.506,Z 1525.160,A 0.000,B 0.000,C 90.000,E1 64.845} C_DIS
LIN {X 0.126,Y -584.823,Z 1525.148,A 0.000,B 0.000,C 90.000,E1 62.666} C_DIS
LIN {X 0.152,Y -585.583,Z 1525.142,A 0.000,B 0.000,C 90.000,E1 61.591} C_DIS
LIN {X -0.057,Y -586.355,Z 1525.136,A 0.000,B 0.000,C 90.000,E1 60.539} C_DIS
LIN {X -0.080,Y -587.336,Z 1525.129,A 0.000,B 0.000,C 90.000,E1 59.203} C_DIS
LIN {X -0.084,Y -588.239,Z 1525.121,A 0.000,B 0.000,C 90.000,E1 57.867} C_DIS
LIN {X 0.239,Y -589.157,Z 1525.114,A 0.000,B 0.000,C 90.000,E1 56.501} C_DIS
LIN {X 0.089,Y -590.080,Z 1525.107,A 0.000,B 0.000,C 90.000,E1 55.182} C_DIS
